LIN {X 0,Y 396.869,Z 754.99,A -85,B 0,C 180,E1 -11238.248,E2 -11238.248} C_VEL
LIN {X 0,Y 396.346,Z 761.62,A -85,B 0,C 180,E1 -11239.785,E2 -11239.785} C_VEL
LIN {X 0,Y 396.097,Z 767.09,A -85,B 0,C 180,E1 -11241.324,E2 -11241.324} C_VEL
LIN {X 0,Y 395.954,Z 771.54,A -85,B 0,C 180,E1 -11242.861,E2 -11242.861} C_VEL
LIN {X 0,Y 395.896,Z 776.01,A -85,B 0,C 180,E1 -11244.906,E2 -11244.906} C_VEL
LIN {X 0,Y 395.865,Z 778.941,A -85,B 0,C 180,E1 -11246.946,E2 -11246.946} C_VEL
LIN {X 0,Y 395.918,Z 779.858,A -85,B 0,C 180,E1 -11247.964,E2 -11247.964} C_VEL
LIN {X 0,Y 395.862,Z 780.59,A -85,B 0,C 180,E1 -11249.999,E2 -11249.999} C_VEL
LIN {X 0,Y 395.918,Z 779.857,A -85,B 0,C 180,E1 -11252.033,E2 -11252.033} C_VEL
LIN {X 0,Y 395.821,Z 777.659,A -85,B 0,C 180,E1 -11254.071,E2 -11254.071} C_VEL
LIN {X 0,Y 395.873,Z 775.066,A -85,B 0,C 180,E1 -11255.602,E2 -11255.602} C_VEL
LIN {X 0,Y 395.952,Z 771.533,A -85,B 0,C 180,E1 -11257.136,E2 -11257.136} C_VEL
LIN {X 0,Y 396.164,Z 765.395,A -85,B 0,C 180,E1 -11259.186,E2 -11259.186} C_VEL
LIN {X 0,Y 396.601,Z 758.452,A -85,B 0,C 180,E1 -11260.98,E2 -11260.98} C_VEL
LIN {X 0,Y 397.107,Z 751.156,A -85,B 0,C 180,E1 -11262.52,E2 -11262.52} C_VEL
LIN {X 0,Y 397.762,Z 742.533,A -85,B 0,C 180,E1 -11264.033,E2 -11264.033} C_VEL
LIN {X 0,Y 398.669,Z 731.702,A -85,B 0,C 180,E1 -11265.594,E2 -11265.594} C_VEL
LIN {X 0,Y 399.641,Z 720.961,A -85,B 0,C 180,E1 -11266.866,E2 -11266.866} C_VEL
LIN {X 0,Y 400.621,Z 709.248,A -85,B 0,C 180,E1 -11268.009,E2 -11268.009} C_VEL
LIN {X 0,Y 401.651,Z 696.152,A -85,B 0,C 180,E1 -11269.036,E2 -11269.036} C_VEL
LIN {X 0,Y 402.545,Z 683.072,A -85,B 0,C 180,E1 -11269.836,E2 -11269.836} C_VEL
LIN {X 0,Y 403.393,Z 668.569,A -85,B 0,C 180,E1 -11270.49,E2 -11270.49} C_VEL
LIN {X 0,Y 404.043,Z 653.982,A -85,B 0,C 180,E1 -11270.922,E2 -11270.922} C_VEL
LIN {X 0,Y 405.933,Z 549.182,A -85,B 0,C 180,E1 -11272.925,E2 -11272.925} C_VEL
LIN {X 0,Y 402.002,Z 522.148,A -85,B 0,C 180,E1 -11273.708,E2 -11273.708} C_VEL
LIN {X 0,Y 403.986,Z 502.582,A -85,B 0,C 180,E1 -11276.89,E2 -11276.89} C_VEL
LIN {X 0,Y 403.831,Z 499.437,A -85,B 0,C 180,E1 -11277.431,E2 -11277.431} C_VEL
LIN {X 0,Y 400.668,Z 486.023,A -85,B 0,C 180,E1 -11279.97,E2 -11279.97} C_VEL
LIN {X 0,Y 397.108,Z 472.647,A -85,B 0,C 180,E1 -11282.667,E2 -11282.667} C_VEL
LIN {X 0,Y 397.103,Z 472.629,A -85,B 0,C 180,E1 -11285.733,E2 -11285.733} C_VEL
LIN {X 0,Y 397.11,Z 472.644,A -85,B 0,C 180,E1 -11289.575,E2 -11289.575} C_VEL
LIN {X 0,Y 397.151,Z 472.639,A -85,B 0,C 180,E1 -11292.254,E2 -11292.254} C_VEL
LIN {X 0,Y 397.143,Z 472.639,A -85,B 0,C 180,E1 -11295.058,E2 -11295.058} C_VEL
LIN {X 0,Y 397.148,Z 472.634,A -85,B 0,C 180,E1 -11298.005,E2 -11298.005} C_VEL
LIN {X 0,Y 397.101,Z 472.639,A -85,B 0,C 180,E1 -11301.725,E2 -11301.725} C_VEL
LIN {X 0,Y 397.116,Z 472.634,A -85,B 0,C 180,E1 -11305.506,E2 -11305.506} C_VEL
LIN {X 0,Y 397.078,Z 472.645,A -85,B 0,C 180,E1 -11309.118,E2 -11309.118} C_VEL
LIN {X 0,Y 397.184,Z 472.632,A -85,B 0,C 180,E1 -11312.609,E2 -11312.609} C_VEL
LIN {X 0,Y 397.122,Z 472.637,A -85,B 0,C 180,E1 -11315.981,E2 -11315.981} C_VEL
LIN {X 0,Y 397.127,Z 472.63,A -85,B 0,C 180,E1 -11319.704,E2 -11319.704} C_VEL
LIN {X 0,Y 397.17,Z 472.635,A -85,B 0,C 180,E1 -11322.844,E2 -11322.844} C_VEL
LIN {X 0,Y 397.215,Z 472.633,A -85,B 0,C 180,E1 -11326.679,E2 -11326.679} C_VEL
LIN {X 0,Y 397.219,Z 472.625,A -85,B 0,C 180,E1 -11329.809,E2 -11329.809} C_VEL
LIN {X 0,Y 397.353,Z 472.606,A -85,B 0,C 180,E1 -11332.888,E2 -11332.888} C_VEL
LIN {X 0,Y 397.247,Z 472.628,A -85,B 0,C 180,E1 -11334.925,E2 -11334.925} C_VEL
LIN {X 0,Y 397.441,Z 472.598,A -85,B 0,C 180,E1 -11337.973,E2 -11337.973} C_VEL
LIN {X 0,Y 397.571,Z 472.582,A -85,B 0,C 180,E1 -11340,E2 -11340} C_VEL
LIN {X 0,Y 397.372,Z 472.602,A -85,B 0,C 180,E1 -11343.042,E2 -11343.042} C_VEL
LIN {X 0,Y 397.352,Z 472.609,A -85,B 0,C 180,E1 -11347.112,E2 -11347.112} C_VEL
LIN {X 0,Y 397.218,Z 472.628,A -85,B 0,C 180,E1 -11350.191,E2 -11350.191} C_VEL
LIN {X 0,Y 397.215,Z 472.622,A -85,B 0,C 180,E1 -11353.322,E2 -11353.322} C_VEL
LIN {X 0,Y 397.16,Z 472.639,A -85,B 0,C 180,E1 -11356.447,E2 -11356.447} C_VEL
LIN {X 0,Y 397.138,Z 472.638,A -85,B 0,C 180,E1 -11359.648,E2 -11359.648} C_VEL
LIN {X 0,Y 397.125,Z 472.64,A -85,B 0,C 180,E1 -11363.041,E2 -11363.041} C_VEL
LIN {X 0,Y 397.125,Z 472.639,A -85,B 0,C 180,E1 -11366.259,E2 -11366.259} C_VEL
LIN {X 0,Y 397.118,Z 472.645,A -85,B 0,C 180,E1 -11368.544,E2 -11368.544} C_VEL
LIN {X 0,Y 397.103,Z 472.644,A -85,B 0,C 180,E1 -11372.07,E2 -11372.07} C_VEL
LIN {X 0,Y 397.112,Z 472.642,A -85,B 0,C 180,E1 -11375.505,E2 -11375.505} C_VEL
LIN {X 0,Y 397.13,Z 472.643,A -85,B 0,C 180,E1 -11378.864,E2 -11378.864} C_VEL
LIN {X 0,Y 397.107,Z 472.648,A -85,B 0,C 180,E1 -11382.263,E2 -11382.263} C_VEL
LIN {X 0,Y 397.159,Z 472.639,A -85,B 0,C 180,E1 -11386.362,E2 -11386.362} C_VEL
LIN {X 0,Y 397.119,Z 472.642,A -85,B 0,C 180,E1 -11389.552,E2 -11389.552} C_VEL
LIN {X 0,Y 397.095,Z 472.637,A -85,B 0,C 180,E1 -11392.791,E2 -11392.791} C_VEL
LIN {X 0,Y 397.115,Z 472.638,A -85,B 0,C 180,E1 -11396.283,E2 -11396.283} C_VEL
LIN {X 0,Y 397.141,Z 472.768,A -85,B 0,C 180,E1 -11399.814,E2 -11399.814} C_VEL
LIN {X 0,Y 400.185,Z 485.268,A -85,B 0,C 180,E1 -11402.833,E2 -11402.833} C_VEL
LIN {X 0,Y 402.101,Z 495.614,A -85,B 0,C 180,E1 -11405.2,E2 -11405.2} C_VEL
LIN {X 0,Y 401.021,Z 508.757,A -85,B 0,C 180,E1 -11407.867,E2 -11407.867} C_VEL
LIN {X 0,Y 400.417,Z 516.355,A -85,B 0,C 180,E1 -11409.385,E2 -11409.385} C_VEL
LIN {X 0,Y 405.174,Z 540.917,A -85,B 0,C 180,E1 -11410.097,E2 -11410.097} C_VEL
LIN {X 0,Y 404.272,Z 629.333,A -85,B 0,C 180,E1 -11411.57,E2 -11411.57} C_VEL
LIN {X 0,Y 403.876,Z 642.226,A -85,B 0,C 180,E1 -11411.977,E2 -11411.977} C_VEL
LIN {X 0,Y 403.222,Z 654.725,A -85,B 0,C 180,E1 -11412.57,E2 -11412.57} C_VEL
LIN {X 0,Y 402.549,Z 665.462,A -85,B 0,C 180,E1 -11413.259,E2 -11413.259} C_VEL
LIN {X 0,Y 401.772,Z 675.831,A -85,B 0,C 180,E1 -11414.106,E2 -11414.106} C_VEL
LIN {X 0,Y 400.872,Z 686.063,A -85,B 0,C 180,E1 -11415.145,E2 -11415.145} C_VEL
LIN {X 0,Y 399.93,Z 695.158,A -85,B 0,C 180,E1 -11416.278,E2 -11416.278} C_VEL
LIN {X 0,Y 399.111,Z 703.472,A -85,B 0,C 180,E1 -11417.544,E2 -11417.544} C_VEL
LIN {X 0,Y 398.218,Z 711.583,A -85,B 0,C 180,E1 -11419.065,E2 -11419.065} C_VEL
LIN {X 0,Y 397.331,Z 719.107,A -85,B 0,C 180,E1 -11420.841,E2 -11420.841} C_VEL
LIN {X 0,Y 396.808,Z 724.17,A -85,B 0,C 180,E1 -11422.368,E2 -11422.368} C_VEL
LIN {X 0,Y 396.438,Z 728.134,A -85,B 0,C 180,E1 -11423.895,E2 -11423.895} C_VEL
LIN {X 0,Y 396.211,Z 730.253,A -85,B 0,C 180,E1 -11424.913,E2 -11424.913} C_VEL
LIN {X 0,Y 396.23,Z 731.923,A -85,B 0,C 180,E1 -11425.933,E2 -11425.933} C_VEL
LIN {X 0,Y 395.984,Z 734.125,A -85,B 0,C 180,E1 -11427.967,E2 -11427.967} C_VEL
LIN {X 0,Y 395.877,Z 734.902,A -85,B 0,C 180,E1 -11430.001,E2 -11430.001} C_VEL
LIN {X 0,Y 395.988,Z 734.15,A -85,B 0,C 180,E1 -11432.085,E2 -11432.085} C_VEL
LIN {X 0,Y 395.386,Z 733.489,A -85,B 0,C 180,E1 -11432.928,E2 -11432.928} C_VEL
LIN {X 0,Y 392.639,Z 732.001,A -85,B 0,C 180,E1 -11434.296,E2 -11434.296} C_VEL
LIN {X 0,Y 390.363,Z 730.358,A -85,B 0,C 180,E1 -11435.388,E2 -11435.388} C_VEL
LIN {X 0,Y 389.488,Z 728.759,A -85,B 0,C 180,E1 -11436.217,E2 -11436.217} C_VEL
LIN {X 0,Y 389.473,Z 728.134,A -85,B 0,C 180,E1 -11436.494,E2 -11436.494} C_VEL
LIN {X 0,Y 389.917,Z 723.331,A -85,B 0,C 180,E1 -11438.292,E2 -11438.292} C_VEL
LIN {X 0,Y 390.69,Z 716.937,A -85,B 0,C 180,E1 -11440.103,E2 -11440.103} C_VEL
LIN {X 0,Y 391.491,Z 709.979,A -85,B 0,C 180,E1 -11441.653,E2 -11441.653} C_VEL
LIN {X 0,Y 392.369,Z 701.359,A -85,B 0,C 180,E1 -11443.203,E2 -11443.203} C_VEL
LIN {X 0,Y 393.541,Z 691.551,A -85,B 0,C 180,E1 -11444.612,E2 -11444.612} C_VEL
LIN {X 0,Y 394.567,Z 680.463,A -85,B 0,C 180,E1 -11445.877,E2 -11445.877} C_VEL
LIN {X 0,Y 395.596,Z 668.922,A -85,B 0,C 180,E1 -11446.914,E2 -11446.914} C_VEL
LIN {X 0,Y 396.493,Z 657.025,A -85,B 0,C 180,E1 -11447.739,E2 -11447.739} C_VEL
LIN {X 0,Y 397.148,Z 644.521,A -85,B 0,C 180,E1 -11448.375,E2 -11448.375} C_VEL
LIN {X 0,Y 397.611,Z 631.502,A -85,B 0,C 180,E1 -11448.82,E2 -11448.82} C_VEL
LIN {X 0,Y 397.959,Z 606.83,A -85,B 0,C 180,E1 -11449.271,E2 -11449.271} C_VEL
LIN {X 0,Y 398.517,Z 540.974,A -85,B 0,C 180,E1 -11450.379,E2 -11450.379} C_VEL
LIN {X 0,Y 393.657,Z 516.432,A -85,B 0,C 180,E1 -11451.114,E2 -11451.114} C_VEL
LIN {X 0,Y 394.865,Z 501.461,A -85,B 0,C 180,E1 -11454.166,E2 -11454.166} C_VEL
LIN {X 0,Y 395.161,Z 496.26,A -85,B 0,C 180,E1 -11455.269,E2 -11455.269} C_VEL
LIN {X 0,Y 392.732,Z 484.528,A -85,B 0,C 180,E1 -11458.035,E2 -11458.035} C_VEL
LIN {X 0,Y 390.068,Z 473.528,A -85,B 0,C 180,E1 -11460.785,E2 -11460.785} C_VEL
LIN {X 0,Y 390.074,Z 473.52,A -85,B 0,C 180,E1 -11464.025,E2 -11464.025} C_VEL
LIN {X 0,Y 390.052,Z 473.527,A -85,B 0,C 180,E1 -11467.552,E2 -11467.552} C_VEL
LIN {X 0,Y 390.064,Z 473.52,A -85,B 0,C 180,E1 -11470.822,E2 -11470.822} C_VEL
LIN {X 0,Y 390.063,Z 473.518,A -85,B 0,C 180,E1 -11473.887,E2 -11473.887} C_VEL
LIN {X 0,Y 390.063,Z 473.52,A -85,B 0,C 180,E1 -11476.79,E2 -11476.79} C_VEL
LIN {X 0,Y 390.062,Z 473.523,A -85,B 0,C 180,E1 -11479.561,E2 -11479.561} C_VEL
LIN {X 0,Y 390.05,Z 473.516,A -85,B 0,C 180,E1 -11482.449,E2 -11482.449} C_VEL
LIN {X 0,Y 390.091,Z 473.52,A -85,B 0,C 180,E1 -11486.047,E2 -11486.047} C_VEL
LIN {X 0,Y 390.053,Z 473.526,A -85,B 0,C 180,E1 -11489.869,E2 -11489.869} C_VEL
LIN {X 0,Y 390.126,Z 473.597,A -85,B 0,C 180,E1 -11490.415,E2 -11490.415} C_VEL
LIN {X 0,Y 393.506,Z 488.852,A -85,B 0,C 180,E1 -11493.254,E2 -11493.254} C_VEL
LIN {X 0,Y 394.678,Z 495.242,A -85,B 0,C 180,E1 -11494.417,E2 -11494.417} C_VEL
LIN {X 0,Y 393.714,Z 514.791,A -85,B 0,C 180,E1 -11497.708,E2 -11497.708} C_VEL
LIN {X 0,Y 393.02,Z 529.732,A -85,B 0,C 180,E1 -11500.217,E2 -11500.217} C_VEL
LIN {X 0,Y 396.012,Z 549.691,A -85,B 0,C 180,E1 -11500.823,E2 -11500.823} C_VEL
LIN {X 0,Y 394.038,Z 641.02,A -85,B 0,C 180,E1 -11502.885,E2 -11502.885} C_VEL
LIN {X 0,Y 393.714,Z 653.198,A -85,B 0,C 180,E1 -11503.338,E2 -11503.338} C_VEL
LIN {X 0,Y 393.126,Z 666.44,A -85,B 0,C 180,E1 -11504.046,E2 -11504.046} C_VEL
LIN {X 0,Y 392.539,Z 677.977,A -85,B 0,C 180,E1 -11504.86,E2 -11504.86} C_VEL
LIN {X 0,Y 391.975,Z 688.733,A -85,B 0,C 180,E1 -11505.823,E2 -11505.823} C_VEL
LIN {X 0,Y 391.293,Z 699.539,A -85,B 0,C 180,E1 -11507.026,E2 -11507.026} C_VEL
LIN {X 0,Y 390.633,Z 709.04,A -85,B 0,C 180,E1 -11508.322,E2 -11508.322} C_VEL
LIN {X 0,Y 390.037,Z 718.2,A -85,B 0,C 180,E1 -11509.881,E2 -11509.881} C_VEL
LIN {X 0,Y 389.558,Z 725.574,A -85,B 0,C 180,E1 -11511.44,E2 -11511.44} C_VEL
LIN {X 0,Y 389.267,Z 730.534,A -85,B 0,C 180,E1 -11512.739,E2 -11512.739} C_VEL
LIN {X 0,Y 389.075,Z 735.328,A -85,B 0,C 180,E1 -11514.298,E2 -11514.298} C_VEL
LIN {X 0,Y 388.873,Z 738.948,A -85,B 0,C 180,E1 -11515.854,E2 -11515.854} C_VEL
LIN {X 0,Y 388.855,Z 740.743,A -85,B 0,C 180,E1 -11516.892,E2 -11516.892} C_VEL
LIN {X 0,Y 388.834,Z 742.115,A -85,B 0,C 180,E1 -11517.928,E2 -11517.928} C_VEL
LIN {X 0,Y 388.767,Z 743.07,A -85,B 0,C 180,E1 -11518.964,E2 -11518.964} C_VEL
LIN {X 0,Y 388.748,Z 743.551,A -85,B 0,C 180,E1 -11520,E2 -11520} C_VEL
LIN {X 0,Y 388.787,Z 743.621,A -85,B 0,C 180,E1 -11521.036,E2 -11521.036} C_VEL
LIN {X 0,Y 388.874,Z 743.279,A -85,B 0,C 180,E1 -11522.071,E2 -11522.071} C_VEL
LIN {X 0,Y 389.015,Z 742.463,A -85,B 0,C 180,E1 -11523.107,E2 -11523.107} C_VEL
LIN {X 0,Y 389.091,Z 741.23,A -85,B 0,C 180,E1 -11524.143,E2 -11524.143} C_VEL
LIN {X 0,Y 389.194,Z 738.55,A -85,B 0,C 180,E1 -11525.7,E2 -11525.7} C_VEL
LIN {X 0,Y 389.568,Z 734.781,A -85,B 0,C 180,E1 -11527.255,E2 -11527.255} C_VEL
LIN {X 0,Y 389.993,Z 729.855,A -85,B 0,C 180,E1 -11528.811,E2 -11528.811} C_VEL
LIN {X 0,Y 390.649,Z 723.594,A -85,B 0,C 180,E1 -11530.364,E2 -11530.364} C_VEL
LIN {X 0,Y 391.342,Z 715.749,A -85,B 0,C 180,E1 -11531.919,E2 -11531.919} C_VEL
LIN {X 0,Y 392.056,Z 707.734,A -85,B 0,C 180,E1 -11533.212,E2 -11533.212} C_VEL
LIN {X 0,Y 392.976,Z 697.935,A -85,B 0,C 180,E1 -11534.5,E2 -11534.5} C_VEL
LIN {X 0,Y 394.037,Z 685.631,A -85,B 0,C 180,E1 -11535.783,E2 -11535.783} C_VEL
LIN {X 0,Y 394.787,Z 674.799,A -85,B 0,C 180,E1 -11536.682,E2 -11536.682} C_VEL
LIN {X 0,Y 395.579,Z 662.942,A -85,B 0,C 180,E1 -11537.446,E2 -11537.446} C_VEL
LIN {X 0,Y 396.221,Z 649.645,A -85,B 0,C 180,E1 -11538.084,E2 -11538.084} C_VEL
LIN {X 0,Y 396.743,Z 635.325,A -85,B 0,C 180,E1 -11538.527,E2 -11538.527} C_VEL
LIN {X 0,Y 399.017,Z 569.961,A -85,B 0,C 180,E1 -11540.177,E2 -11540.177} C_VEL
LIN {X 0,Y 399.7,Z 550.541,A -85,B 0,C 180,E1 -11540.697,E2 -11540.697} C_VEL
LIN {X 0,Y 397.165,Z 537.555,A -85,B 0,C 180,E1 -11541.299,E2 -11541.299} C_VEL
LIN {X 0,Y 396.171,Z 533.316,A -85,B 0,C 180,E1 -11541.53,E2 -11541.53} C_VEL
LIN {X 0,Y 397.739,Z 510.589,A -85,B 0,C 180,E1 -11545.379,E2 -11545.379} C_VEL
LIN {X 0,Y 398.225,Z 502.569,A -85,B 0,C 180,E1 -11546.746,E2 -11546.746} C_VEL
LIN {X 0,Y 397.063,Z 495.233,A -85,B 0,C 180,E1 -11548.217,E2 -11548.217} C_VEL
LIN {X 0,Y 394.529,Z 486.198,A -85,B 0,C 180,E1 -11550.183,E2 -11550.183} C_VEL
LIN {X 0,Y 391.296,Z 476.89,A -85,B 0,C 180,E1 -11552.416,E2 -11552.416} C_VEL
LIN {X 0,Y 390.097,Z 473.519,A -85,B 0,C 180,E1 -11553.332,E2 -11553.332} C_VEL
LIN {X 0,Y 390.065,Z 473.525,A -85,B 0,C 180,E1 -11556.483,E2 -11556.483} C_VEL
LIN {X 0,Y 390.077,Z 473.52,A -85,B 0,C 180,E1 -11559.218,E2 -11559.218} C_VEL
LIN {X 0,Y 390.047,Z 473.525,A -85,B 0,C 180,E1 -11562.373,E2 -11562.373} C_VEL
LIN {X 0,Y 390.049,Z 473.523,A -85,B 0,C 180,E1 -11565.354,E2 -11565.354} C_VEL
LIN {X 0,Y 390.036,Z 473.526,A -85,B 0,C 180,E1 -11568.186,E2 -11568.186} C_VEL
LIN {X 0,Y 390.092,Z 473.515,A -85,B 0,C 180,E1 -11570.907,E2 -11570.907} C_VEL
LIN {X 0,Y 390.089,Z 473.52,A -85,B 0,C 180,E1 -11574.792,E2 -11574.792} C_VEL
LIN {X 0,Y 390.078,Z 473.534,A -85,B 0,C 180,E1 -11576.858,E2 -11576.858} C_VEL
LIN {X 0,Y 394.193,Z 489.099,A -85,B 0,C 180,E1 -11580.051,E2 -11580.051} C_VEL
LIN {X 0,Y 396.925,Z 500.672,A -85,B 0,C 180,E1 -11582.289,E2 -11582.289} C_VEL
LIN {X 0,Y 397.307,Z 502.415,A -85,B 0,C 180,E1 -11582.617,E2 -11582.617} C_VEL
LIN {X 0,Y 395.596,Z 519.085,A -85,B 0,C 180,E1 -11585.378,E2 -11585.378} C_VEL
LIN {X 0,Y 395.25,Z 522.317,A -85,B 0,C 180,E1 -11585.915,E2 -11585.915} C_VEL
LIN {X 0,Y 399.311,Z 550.056,A -85,B 0,C 180,E1 -11586.712,E2 -11586.712} C_VEL
LIN {X 0,Y 397.368,Z 652.886,A -85,B 0,C 180,E1 -11588.707,E2 -11588.707} C_VEL
LIN {X 0,Y 396.788,Z 666.902,A -85,B 0,C 180,E1 -11589.116,E2 -11589.116} C_VEL
LIN {X 0,Y 395.894,Z 681.293,A -85,B 0,C 180,E1 -11589.746,E2 -11589.746} C_VEL
LIN {X 0,Y 394.988,Z 694.805,A -85,B 0,C 180,E1 -11590.566,E2 -11590.566} C_VEL
LIN {X 0,Y 394.005,Z 707.301,A -85,B 0,C 180,E1 -11591.541,E2 -11591.541} C_VEL
LIN {X 0,Y 392.907,Z 719.288,A -85,B 0,C 180,E1 -11592.699,E2 -11592.699} C_VEL
LIN {X 0,Y 391.778,Z 731.243,A -85,B 0,C 180,E1 -11594.122,E2 -11594.122} C_VEL
LIN {X 0,Y 390.79,Z 742.088,A -85,B 0,C 180,E1 -11595.709,E2 -11595.709} C_VEL
LIN {X 0,Y 390.155,Z 750.762,A -85,B 0,C 180,E1 -11597.258,E2 -11597.258} C_VEL
LIN {X 0,Y 389.473,Z 759.092,A -85,B 0,C 180,E1 -11599.077,E2 -11599.077} C_VEL
LIN {X 0,Y 389.098,Z 764.977,A -85,B 0,C 180,E1 -11600.643,E2 -11600.643} C_VEL
LIN {X 0,Y 388.896,Z 769.755,A -85,B 0,C 180,E1 -11602.209,E2 -11602.209} C_VEL
LIN {X 0,Y 388.789,Z 774.38,A -85,B 0,C 180,E1 -11604.157,E2 -11604.157} C_VEL
LIN {X 0,Y 388.745,Z 777.246,A -85,B 0,C 180,E1 -11605.852,E2 -11605.852} C_VEL
LIN {X 0,Y 388.849,Z 779.449,A -85,B 0,C 180,E1 -11607.927,E2 -11607.927} C_VEL
LIN {X 0,Y 388.787,Z 780.181,A -85,B 0,C 180,E1 -11609.999,E2 -11609.999} C_VEL
LIN {X 0,Y 388.848,Z 779.448,A -85,B 0,C 180,E1 -11612.07,E2 -11612.07} C_VEL
LIN {X 0,Y 388.744,Z 777.246,A -85,B 0,C 180,E1 -11614.146,E2 -11614.146} C_VEL
LIN {X 0,Y 388.788,Z 774.375,A -85,B 0,C 180,E1 -11615.841,E2 -11615.841} C_VEL
LIN {X 0,Y 388.893,Z 769.744,A -85,B 0,C 180,E1 -11617.788,E2 -11617.788} C_VEL
LIN {X 0,Y 389.095,Z 764.964,A -85,B 0,C 180,E1 -11619.354,E2 -11619.354} C_VEL
LIN {X 0,Y 389.573,Z 758.009,A -85,B 0,C 180,E1 -11621.181,E2 -11621.181} C_VEL
LIN {X 0,Y 390.177,Z 749.536,A -85,B 0,C 180,E1 -11622.968,E2 -11622.968} C_VEL
LIN {X 0,Y 390.963,Z 740.229,A -85,B 0,C 180,E1 -11624.575,E2 -11624.575} C_VEL
LIN {X 0,Y 391.792,Z 731.211,A -85,B 0,C 180,E1 -11625.874,E2 -11625.874} C_VEL
LIN {X 0,Y 392.807,Z 720.442,A -85,B 0,C 180,E1 -11627.169,E2 -11627.169} C_VEL
LIN {X 0,Y 393.838,Z 708.693,A -85,B 0,C 180,E1 -11628.33,E2 -11628.33} C_VEL
LIN {X 0,Y 394.87,Z 695.851,A -85,B 0,C 180,E1 -11629.352,E2 -11629.352} C_VEL
LIN {X 0,Y 395.862,Z 682.385,A -85,B 0,C 180,E1 -11630.185,E2 -11630.185} C_VEL
LIN {X 0,Y 396.733,Z 667.646,A -85,B 0,C 180,E1 -11630.85,E2 -11630.85} C_VEL
LIN {X 0,Y 397.344,Z 654.089,A -85,B 0,C 180,E1 -11631.258,E2 -11631.258} C_VEL
LIN {X 0,Y 399.311,Z 549.835,A -85,B 0,C 180,E1 -11633.282,E2 -11633.282} C_VEL
LIN {X 0,Y 395.271,Z 522.131,A -85,B 0,C 180,E1 -11634.099,E2 -11634.099} C_VEL
LIN {X 0,Y 397.21,Z 504.027,A -85,B 0,C 180,E1 -11637.102,E2 -11637.102} C_VEL
LIN {X 0,Y 396.904,Z 500.649,A -85,B 0,C 180,E1 -11637.705,E2 -11637.705} C_VEL
LIN {X 0,Y 393.389,Z 485.818,A -85,B 0,C 180,E1 -11640.585,E2 -11640.585} C_VEL
LIN {X 0,Y 390.072,Z 473.522,A -85,B 0,C 180,E1 -11643.178,E2 -11643.178} C_VEL
LIN {X 0,Y 390.054,Z 473.517,A -85,B 0,C 180,E1 -11646.482,E2 -11646.482} C_VEL
LIN {X 0,Y 390.068,Z 473.52,A -85,B 0,C 180,E1 -11649.218,E2 -11649.218} C_VEL
LIN {X 0,Y 390.113,Z 473.516,A -85,B 0,C 180,E1 -11652.385,E2 -11652.385} C_VEL
LIN {X 0,Y 390.121,Z 473.511,A -85,B 0,C 180,E1 -11656.101,E2 -11656.101} C_VEL
LIN {X 0,Y 390.07,Z 473.515,A -85,B 0,C 180,E1 -11659.562,E2 -11659.562} C_VEL
LIN {X 0,Y 390.038,Z 473.518,A -85,B 0,C 180,E1 -11662.447,E2 -11662.447} C_VEL
LIN {X 0,Y 390.058,Z 473.514,A -85,B 0,C 180,E1 -11666.044,E2 -11666.044} C_VEL
LIN {X 0,Y 390.038,Z 473.521,A -85,B 0,C 180,E1 -11668.497,E2 -11668.497} C_VEL
LIN {X 0,Y 390.107,Z 473.512,A -85,B 0,C 180,E1 -11672.069,E2 -11672.069} C_VEL
LIN {X 0,Y 390.069,Z 473.515,A -85,B 0,C 180,E1 -11675.519,E2 -11675.519} C_VEL
LIN {X 0,Y 390.044,Z 473.503,A -85,B 0,C 180,E1 -11678.877,E2 -11678.877} C_VEL
LIN {X 0,Y 390.117,Z 473.515,A -85,B 0,C 180,E1 -11682.166,E2 -11682.166} C_VEL
LIN {X 0,Y 390.136,Z 473.51,A -85,B 0,C 180,E1 -11685.392,E2 -11685.392} C_VEL
LIN {X 0,Y 390.15,Z 473.506,A -85,B 0,C 180,E1 -11688.571,E2 -11688.571} C_VEL
LIN {X 0,Y 390.332,Z 473.487,A -85,B 0,C 180,E1 -11691.993,E2 -11691.993} C_VEL
LIN {X 0,Y 390.219,Z 473.502,A -85,B 0,C 180,E1 -11694.834,E2 -11694.834} C_VEL
LIN {X 0,Y 390.41,Z 473.473,A -85,B 0,C 180,E1 -11697.937,E2 -11697.937} C_VEL
LIN {X 0,Y 390.541,Z 473.458,A -85,B 0,C 180,E1 -11700,E2 -11700} C_VEL
LIN {X 0,Y 390.306,Z 473.482,A -85,B 0,C 180,E1 -11703.097,E2 -11703.097} C_VEL
LIN {X 0,Y 390.298,Z 473.489,A -85,B 0,C 180,E1 -11706.653,E2 -11706.653} C_VEL
LIN {X 0,Y 390.199,Z 473.5,A -85,B 0,C 180,E1 -11709.329,E2 -11709.329} C_VEL
LIN {X 0,Y 390.167,Z 473.505,A -85,B 0,C 180,E1 -11712.483,E2 -11712.483} C_VEL
LIN {X 0,Y 390.134,Z 473.511,A -85,B 0,C 180,E1 -11715.677,E2 -11715.677} C_VEL
LIN {X 0,Y 390.095,Z 473.518,A -85,B 0,C 180,E1 -11718.923,E2 -11718.923} C_VEL
LIN {X 0,Y 390.03,Z 473.521,A -85,B 0,C 180,E1 -11722.235,E2 -11722.235} C_VEL
LIN {X 0,Y 390.109,Z 473.512,A -85,B 0,C 180,E1 -11725.744,E2 -11725.744} C_VEL
LIN {X 0,Y 390.056,Z 473.519,A -85,B 0,C 180,E1 -11729.11,E2 -11729.11} C_VEL
LIN {X 0,Y 390.047,Z 473.522,A -85,B 0,C 180,E1 -11732.721,E2 -11732.721} C_VEL
LIN {X 0,Y 390.049,Z 473.523,A -85,B 0,C 180,E1 -11735.827,E2 -11735.827} C_VEL
LIN {X 0,Y 390.067,Z 473.52,A -85,B 0,C 180,E1 -11739.221,E2 -11739.221} C_VEL
LIN {X 0,Y 390.073,Z 473.523,A -85,B 0,C 180,E1 -11742.382,E2 -11742.382} C_VEL
LIN {X 0,Y 390.099,Z 473.516,A -85,B 0,C 180,E1 -11746.107,E2 -11746.107} C_VEL
LIN {X 0,Y 390.078,Z 473.52,A -85,B 0,C 180,E1 -11749.175,E2 -11749.175} C_VEL
LIN {X 0,Y 390.043,Z 473.518,A -85,B 0,C 180,E1 -11752.45,E2 -11752.45} C_VEL
LIN {X 0,Y 390.08,Z 473.514,A -85,B 0,C 180,E1 -11756.048,E2 -11756.048} C_VEL
LIN {X 0,Y 390.072,Z 473.593,A -85,B 0,C 180,E1 -11759.368,E2 -11759.368} C_VEL
LIN {X 0,Y 393.284,Z 486.581,A -85,B 0,C 180,E1 -11762.571,E2 -11762.571} C_VEL
LIN {X 0,Y 395.258,Z 497.309,A -85,B 0,C 180,E1 -11765.07,E2 -11765.07} C_VEL
LIN {X 0,Y 394.135,Z 510.26,A -85,B 0,C 180,E1 -11767.735,E2 -11767.735} C_VEL
LIN {X 0,Y 393.621,Z 516.406,A -85,B 0,C 180,E1 -11768.982,E2 -11768.982} C_VEL
LIN {X 0,Y 398.641,Z 542.404,A -85,B 0,C 180,E1 -11769.752,E2 -11769.752} C_VEL
LIN {X 0,Y 397.624,Z 629.27,A -85,B 0,C 180,E1 -11771.217,E2 -11771.217} C_VEL
LIN {X 0,Y 397.211,Z 642.287,A -85,B 0,C 180,E1 -11771.631,E2 -11771.631} C_VEL
LIN {X 0,Y 396.491,Z 655.415,A -85,B 0,C 180,E1 -11772.264,E2 -11772.264} C_VEL
LIN {X 0,Y 395.722,Z 667.788,A -85,B 0,C 180,E1 -11773.095,E2 -11773.095} C_VEL
LIN {X 0,Y 394.827,Z 678.149,A -85,B 0,C 180,E1 -11773.991,E2 -11773.991} C_VEL
LIN {X 0,Y 393.806,Z 688.712,A -85,B 0,C 180,E1 -11775.137,E2 -11775.137} C_VEL
LIN {X 0,Y 392.625,Z 699.133,A -85,B 0,C 180,E1 -11776.545,E2 -11776.545} C_VEL
LIN {X 0,Y 391.809,Z 706.82,A -85,B 0,C 180,E1 -11777.834,E2 -11777.834} C_VEL
LIN {X 0,Y 390.996,Z 714.39,A -85,B 0,C 180,E1 -11779.385,E2 -11779.385} C_VEL
LIN {X 0,Y 390.12,Z 721.344,A -85,B 0,C 180,E1 -11781.193,E2 -11781.193} C_VEL
LIN {X 0,Y 389.617,Z 726.149,A -85,B 0,C 180,E1 -11782.797,E2 -11782.797} C_VEL
LIN {X 0,Y 389.249,Z 729.655,A -85,B 0,C 180,E1 -11784.302,E2 -11784.302} C_VEL
LIN {X 0,Y 389.145,Z 732.336,A -85,B 0,C 180,E1 -11785.859,E2 -11785.859} C_VEL
LIN {X 0,Y 389.068,Z 733.613,A -85,B 0,C 180,E1 -11786.895,E2 -11786.895} C_VEL
LIN {X 0,Y 388.82,Z 735.099,A -85,B 0,C 180,E1 -11788.966,E2 -11788.966} C_VEL
LIN {X 0,Y 388.82,Z 735.14,A -85,B 0,C 180,E1 -11791.037,E2 -11791.037} C_VEL
LIN {X 0,Y 389.061,Z 733.707,A -85,B 0,C 180,E1 -11793.108,E2 -11793.108} C_VEL
LIN {X 0,Y 389.139,Z 730.838,A -85,B 0,C 180,E1 -11795.182,E2 -11795.182} C_VEL
LIN {X 0,Y 389.473,Z 728.134,A -85,B 0,C 180,E1 -11796.494,E2 -11796.494} C_VEL
LIN {X 0,Y 389.031,Z 726.201,A -85,B 0,C 180,E1 -11797.312,E2 -11797.312} C_VEL
LIN {X 0,Y 386.59,Z 722.711,A -85,B 0,C 180,E1 -11798.634,E2 -11798.634} C_VEL
LIN {X 0,Y 384.23,Z 718.625,A -85,B 0,C 180,E1 -11799.931,E2 -11799.931} C_VEL
LIN {X 0,Y 383.922,Z 715.69,A -85,B 0,C 180,E1 -11800.698,E2 -11800.698} C_VEL
LIN {X 0,Y 384.866,Z 707.784,A -85,B 0,C 180,E1 -11802.391,E2 -11802.391} C_VEL
LIN {X 0,Y 385.694,Z 700.216,A -85,B 0,C 180,E1 -11803.704,E2 -11803.704} C_VEL
LIN {X 0,Y 386.934,Z 689.951,A -85,B 0,C 180,E1 -11805.136,E2 -11805.136} C_VEL
LIN {X 0,Y 387.918,Z 679.348,A -85,B 0,C 180,E1 -11806.33,E2 -11806.33} C_VEL
LIN {X 0,Y 388.974,Z 667.896,A -85,B 0,C 180,E1 -11807.346,E2 -11807.346} C_VEL
LIN {X 0,Y 389.831,Z 656.578,A -85,B 0,C 180,E1 -11808.12,E2 -11808.12} C_VEL
LIN {X 0,Y 390.521,Z 643.778,A -85,B 0,C 180,E1 -11808.766,E2 -11808.766} C_VEL
LIN {X 0,Y 390.991,Z 631.407,A -85,B 0,C 180,E1 -11809.185,E2 -11809.185} C_VEL
LIN {X 0,Y 391.327,Z 604.587,A -85,B 0,C 180,E1 -11809.68,E2 -11809.68} C_VEL
LIN {X 0,Y 391.961,Z 542.061,A -85,B 0,C 180,E1 -11810.746,E2 -11810.746} C_VEL
LIN {X 0,Y 386.872,Z 516.455,A -85,B 0,C 180,E1 -11811.539,E2 -11811.539} C_VEL
LIN {X 0,Y 388.172,Z 501.64,A -85,B 0,C 180,E1 -11814.61,E2 -11814.61} C_VEL
LIN {X 0,Y 388.349,Z 498.091,A -85,B 0,C 180,E1 -11815.379,E2 -11815.379} C_VEL
LIN {X 0,Y 385.846,Z 486.056,A -85,B 0,C 180,E1 -11818.268,E2 -11818.268} C_VEL
LIN {X 0,Y 383.262,Z 475.636,A -85,B 0,C 180,E1 -11820.895,E2 -11820.895} C_VEL
LIN {X 0,Y 383.006,Z 474.406,A -85,B 0,C 180,E1 -11821.225,E2 -11821.225} C_VEL
LIN {X 0,Y 383.024,Z 474.398,A -85,B 0,C 180,E1 -11824.669,E2 -11824.669} C_VEL
LIN {X 0,Y 383.008,Z 474.4,A -85,B 0,C 180,E1 -11827.905,E2 -11827.905} C_VEL
LIN {X 0,Y 382.992,Z 474.4,A -85,B 0,C 180,E1 -11831.348,E2 -11831.348} C_VEL
LIN {X 0,Y 383.004,Z 474.395,A -85,B 0,C 180,E1 -11834.304,E2 -11834.304} C_VEL
LIN {X 0,Y 383.016,Z 474.396,A -85,B 0,C 180,E1 -11837.241,E2 -11837.241} C_VEL
LIN {X 0,Y 383.02,Z 474.397,A -85,B 0,C 180,E1 -11840.414,E2 -11840.414} C_VEL
LIN {X 0,Y 383.033,Z 474.399,A -85,B 0,C 180,E1 -11844.045,E2 -11844.045} C_VEL
LIN {X 0,Y 382.993,Z 474.405,A -85,B 0,C 180,E1 -11847.578,E2 -11847.578} C_VEL
LIN {X 0,Y 383.042,Z 474.439,A -85,B 0,C 180,E1 -11850.127,E2 -11850.127} C_VEL
LIN {X 0,Y 386.482,Z 489.74,A -85,B 0,C 180,E1 -11853.006,E2 -11853.006} C_VEL
LIN {X 0,Y 387.748,Z 496.285,A -85,B 0,C 180,E1 -11854.214,E2 -11854.214} C_VEL
LIN {X 0,Y 386.876,Z 514.365,A -85,B 0,C 180,E1 -11857.292,E2 -11857.292} C_VEL
LIN {X 0,Y 386.116,Z 530.078,A -85,B 0,C 180,E1 -11859.946,E2 -11859.946} C_VEL
LIN {X 0,Y 389.1,Z 551.277,A -85,B 0,C 180,E1 -11860.586,E2 -11860.586} C_VEL
LIN {X 0,Y 387.089,Z 640.853,A -85,B 0,C 180,E1 -11862.67,E2 -11862.67} C_VEL
LIN {X 0,Y 386.737,Z 653.842,A -85,B 0,C 180,E1 -11863.164,E2 -11863.164} C_VEL
LIN {X 0,Y 386.14,Z 666.958,A -85,B 0,C 180,E1 -11863.885,E2 -11863.885} C_VEL
LIN {X 0,Y 385.467,Z 679.541,A -85,B 0,C 180,E1 -11864.806,E2 -11864.806} C_VEL
LIN {X 0,Y 384.796,Z 691.372,A -85,B 0,C 180,E1 -11865.925,E2 -11865.925} C_VEL
LIN {X 0,Y 384.168,Z 701.006,A -85,B 0,C 180,E1 -11867.05,E2 -11867.05} C_VEL
LIN {X 0,Y 383.488,Z 710.257,A -85,B 0,C 180,E1 -11868.37,E2 -11868.37} C_VEL
LIN {X 0,Y 382.916,Z 719.281,A -85,B 0,C 180,E1 -11869.958,E2 -11869.958} C_VEL
LIN {X 0,Y 382.443,Z 726.496,A -85,B 0,C 180,E1 -11871.546,E2 -11871.546} C_VEL
LIN {X 0,Y 382.112,Z 732.811,A -85,B 0,C 180,E1 -11873.319,E2 -11873.319} C_VEL
LIN {X 0,Y 381.944,Z 736.704,A -85,B 0,C 180,E1 -11874.721,E2 -11874.721} C_VEL
LIN {X 0,Y 381.799,Z 739.078,A -85,B 0,C 180,E1 -11875.777,E2 -11875.777} C_VEL
LIN {X 0,Y 381.76,Z 740.938,A -85,B 0,C 180,E1 -11876.834,E2 -11876.834} C_VEL
LIN {X 0,Y 381.753,Z 742.35,A -85,B 0,C 180,E1 -11877.89,E2 -11877.89} C_VEL
LIN {X 0,Y 381.7,Z 743.353,A -85,B 0,C 180,E1 -11878.945,E2 -11878.945} C_VEL
LIN {X 0,Y 381.678,Z 743.888,A -85,B 0,C 180,E1 -11880,E2 -11880} C_VEL
LIN {X 0,Y 381.719,Z 743.99,A -85,B 0,C 180,E1 -11881.055,E2 -11881.055} C_VEL
LIN {X 0,Y 381.813,Z 743.681,A -85,B 0,C 180,E1 -11882.11,E2 -11882.11} C_VEL
LIN {X 0,Y 381.961,Z 742.917,A -85,B 0,C 180,E1 -11883.164,E2 -11883.164} C_VEL
LIN {X 0,Y 382.011,Z 741.714,A -85,B 0,C 180,E1 -11884.22,E2 -11884.22} C_VEL
LIN {X 0,Y 382.161,Z 739.101,A -85,B 0,C 180,E1 -11885.805,E2 -11885.805} C_VEL
LIN {X 0,Y 382.555,Z 735.412,A -85,B 0,C 180,E1 -11887.388,E2 -11887.388} C_VEL
LIN {X 0,Y 383.02,Z 730.554,A -85,B 0,C 180,E1 -11888.973,E2 -11888.973} C_VEL
LIN {X 0,Y 383.712,Z 724.374,A -85,B 0,C 180,E1 -11890.554,E2 -11890.554} C_VEL
LIN {X 0,Y 384.455,Z 716.594,A -85,B 0,C 180,E1 -11892.135,E2 -11892.135} C_VEL
LIN {X 0,Y 385.358,Z 706.949,A -85,B 0,C 180,E1 -11893.715,E2 -11893.715} C_VEL
LIN {X 0,Y 386.482,Z 696.456,A -85,B 0,C 180,E1 -11895.068,E2 -11895.068} C_VEL
LIN {X 0,Y 387.443,Z 685.682,A -85,B 0,C 180,E1 -11896.194,E2 -11896.194} C_VEL
LIN {X 0,Y 388.364,Z 672.938,A -85,B 0,C 180,E1 -11897.237,E2 -11897.237} C_VEL
LIN {X 0,Y 389.181,Z 660.423,A -85,B 0,C 180,E1 -11898.014,E2 -11898.014} C_VEL
LIN {X 0,Y 389.931,Z 645.802,A -85,B 0,C 180,E1 -11898.658,E2 -11898.658} C_VEL
LIN {X 0,Y 391.262,Z 607.662,A -85,B 0,C 180,E1 -11899.682,E2 -11899.682} C_VEL
LIN {X 0,Y 393.514,Z 551.711,A -85,B 0,C 180,E1 -11901.178,E2 -11901.178} C_VEL
LIN {X 0,Y 391.231,Z 539.757,A -85,B 0,C 180,E1 -11901.771,E2 -11901.771} C_VEL
LIN {X 0,Y 389.851,Z 533.727,A -85,B 0,C 180,E1 -11902.112,E2 -11902.112} C_VEL
LIN {X 0,Y 391.439,Z 512.102,A -85,B 0,C 180,E1 -11905.831,E2 -11905.831} C_VEL
LIN {X 0,Y 391.907,Z 504.375,A -85,B 0,C 180,E1 -11907.212,E2 -11907.212} C_VEL
LIN {X 0,Y 390.657,Z 497.292,A -85,B 0,C 180,E1 -11908.68,E2 -11908.68} C_VEL
LIN {X 0,Y 387.868,Z 487.536,A -85,B 0,C 180,E1 -11910.91,E2 -11910.91} C_VEL
LIN {X 0,Y 384.548,Z 478.43,A -85,B 0,C 180,E1 -11913.249,E2 -11913.249} C_VEL
LIN {X 0,Y 383.043,Z 474.397,A -85,B 0,C 180,E1 -11914.403,E2 -11914.403} C_VEL
LIN {X 0,Y 383.007,Z 474.403,A -85,B 0,C 180,E1 -11917.904,E2 -11917.904} C_VEL
LIN {X 0,Y 382.989,Z 474.405,A -85,B 0,C 180,E1 -11921.347,E2 -11921.347} C_VEL
LIN {X 0,Y 383.001,Z 474.404,A -85,B 0,C 180,E1 -11924.303,E2 -11924.303} C_VEL
LIN {X 0,Y 383.015,Z 474.398,A -85,B 0,C 180,E1 -11927.239,E2 -11927.239} C_VEL
LIN {X 0,Y 383.018,Z 474.397,A -85,B 0,C 180,E1 -11930.413,E2 -11930.413} C_VEL
LIN {X 0,Y 383.029,Z 474.397,A -85,B 0,C 180,E1 -11934.044,E2 -11934.044} C_VEL
LIN {X 0,Y 383.052,Z 474.408,A -85,B 0,C 180,E1 -11936.37,E2 -11936.37} C_VEL
LIN {X 0,Y 387.306,Z 490.402,A -85,B 0,C 180,E1 -11939.735,E2 -11939.735} C_VEL
LIN {X 0,Y 390.282,Z 503.153,A -85,B 0,C 180,E1 -11942.249,E2 -11942.249} C_VEL
LIN {X 0,Y 390.464,Z 505.506,A -85,B 0,C 180,E1 -11942.678,E2 -11942.678} C_VEL
LIN {X 0,Y 388.526,Z 522.291,A -85,B 0,C 180,E1 -11945.504,E2 -11945.504} C_VEL
LIN {X 0,Y 392.711,Z 550.453,A -85,B 0,C 180,E1 -11946.336,E2 -11946.336} C_VEL
LIN {X 0,Y 390.671,Z 654.466,A -85,B 0,C 180,E1 -11948.393,E2 -11948.393} C_VEL
LIN {X 0,Y 390.015,Z 668.671,A -85,B 0,C 180,E1 -11948.84,E2 -11948.84} C_VEL
LIN {X 0,Y 389.073,Z 682.935,A -85,B 0,C 180,E1 -11949.513,E2 -11949.513} C_VEL
LIN {X 0,Y 388.024,Z 696.825,A -85,B 0,C 180,E1 -11950.406,E2 -11950.406} C_VEL
LIN {X 0,Y 387.006,Z 709.645,A -85,B 0,C 180,E1 -11951.469,E2 -11951.469} C_VEL
LIN {X 0,Y 385.847,Z 721.167,A -85,B 0,C 180,E1 -11952.646,E2 -11952.646} C_VEL
LIN {X 0,Y 384.692,Z 732.723,A -85,B 0,C 180,E1 -11954.094,E2 -11954.094} C_VEL
LIN {X 0,Y 383.715,Z 743.02,A -85,B 0,C 180,E1 -11955.683,E2 -11955.683} C_VEL
LIN {X 0,Y 383.042,Z 751.56,A -85,B 0,C 180,E1 -11957.279,E2 -11957.279} C_VEL
LIN {X 0,Y 382.354,Z 759.704,A -85,B 0,C 180,E1 -11959.139,E2 -11959.139} C_VEL
LIN {X 0,Y 381.937,Z 766.234,A -85,B 0,C 180,E1 -11961,E2 -11961} C_VEL
LIN {X 0,Y 381.796,Z 770.699,A -85,B 0,C 180,E1 -11962.595,E2 -11962.595} C_VEL
LIN {X 0,Y 381.739,Z 773.456,A -85,B 0,C 180,E1 -11963.807,E2 -11963.807} C_VEL
LIN {X 0,Y 381.67,Z 776.834,A -85,B 0,C 180,E1 -11965.775,E2 -11965.775} C_VEL
LIN {X 0,Y 381.779,Z 779.04,A -85,B 0,C 180,E1 -11967.889,E2 -11967.889} C_VEL
LIN {X 0,Y 381.714,Z 779.773,A -85,B 0,C 180,E1 -11969.999,E2 -11969.999} C_VEL
LIN {X 0,Y 381.779,Z 779.038,A -85,B 0,C 180,E1 -11972.109,E2 -11972.109} C_VEL
LIN {X 0,Y 381.669,Z 776.833,A -85,B 0,C 180,E1 -11974.223,E2 -11974.223} C_VEL
LIN {X 0,Y 381.761,Z 773.134,A -85,B 0,C 180,E1 -11976.34,E2 -11976.34} C_VEL
LIN {X 0,Y 381.89,Z 767.829,A -85,B 0,C 180,E1 -11978.465,E2 -11978.465} C_VEL
LIN {X 0,Y 382.151,Z 762.67,A -85,B 0,C 180,E1 -11980.06,E2 -11980.06} C_VEL
LIN {X 0,Y 382.749,Z 755.255,A -85,B 0,C 180,E1 -11981.92,E2 -11981.92} C_VEL
LIN {X 0,Y 383.403,Z 746.464,A -85,B 0,C 180,E1 -11983.707,E2 -11983.707} C_VEL
LIN {X 0,Y 384.318,Z 736.34,A -85,B 0,C 180,E1 -11985.375,E2 -11985.375} C_VEL
LIN {X 0,Y 385.303,Z 725.568,A -85,B 0,C 180,E1 -11986.83,E2 -11986.83} C_VEL
LIN {X 0,Y 386.57,Z 713.674,A -85,B 0,C 180,E1 -11988.138,E2 -11988.138} C_VEL
LIN {X 0,Y 387.676,Z 700.748,A -85,B 0,C 180,E1 -11989.291,E2 -11989.291} C_VEL
LIN {X 0,Y 388.78,Z 687.334,A -85,B 0,C 180,E1 -11990.224,E2 -11990.224} C_VEL
LIN {X 0,Y 389.7,Z 673.055,A -85,B 0,C 180,E1 -11990.968,E2 -11990.968} C_VEL
LIN {X 0,Y 390.499,Z 658.964,A -85,B 0,C 180,E1 -11991.476,E2 -11991.476} C_VEL
LIN {X 0,Y 390.99,Z 638.331,A -85,B 0,C 180,E1 -11991.932,E2 -11991.932} C_VEL
LIN {X 0,Y 392.682,Z 550.443,A -85,B 0,C 180,E1 -11993.655,E2 -11993.655} C_VEL
LIN {X 0,Y 388.562,Z 522.056,A -85,B 0,C 180,E1 -11994.513,E2 -11994.513} C_VEL
LIN {X 0,Y 390.422,Z 505.448,A -85,B 0,C 180,E1 -11997.322,E2 -11997.322} C_VEL
LIN {X 0,Y 389.986,Z 501.847,A -85,B 0,C 180,E1 -11997.989,E2 -11997.989} C_VEL
LIN {X 0,Y 386.908,Z 488.83,A -85,B 0,C 180,E1 -12000.569,E2 -12000.569} C_VEL
LIN {X 0,Y 383.042,Z 474.387,A -85,B 0,C 180,E1 -12003.628,E2 -12003.628} C_VEL
LIN {X 0,Y 382.993,Z 474.404,A -85,B 0,C 180,E1 -12007.267,E2 -12007.267} C_VEL
LIN {X 0,Y 383.015,Z 474.4,A -85,B 0,C 180,E1 -12009.955,E2 -12009.955} C_VEL
LIN {X 0,Y 383.058,Z 474.397,A -85,B 0,C 180,E1 -12012.787,E2 -12012.787} C_VEL
LIN {X 0,Y 383.064,Z 474.39,A -85,B 0,C 180,E1 -12015.799,E2 -12015.799} C_VEL
LIN {X 0,Y 383.036,Z 474.397,A -85,B 0,C 180,E1 -12018.785,E2 -12018.785} C_VEL
LIN {X 0,Y 382.994,Z 474.398,A -85,B 0,C 180,E1 -12022.094,E2 -12022.094} C_VEL
LIN {X 0,Y 383.009,Z 474.389,A -85,B 0,C 180,E1 -12025.331,E2 -12025.331} C_VEL
LIN {X 0,Y 383.027,Z 474.394,A -85,B 0,C 180,E1 -12027.852,E2 -12027.852} C_VEL
LIN {X 0,Y 383.053,Z 474.39,A -85,B 0,C 180,E1 -12031.72,E2 -12031.72} C_VEL
LIN {X 0,Y 383.041,Z 474.392,A -85,B 0,C 180,E1 -12035.039,E2 -12035.039} C_VEL
LIN {X 0,Y 382.982,Z 474.377,A -85,B 0,C 180,E1 -12038.468,E2 -12038.468} C_VEL
LIN {X 0,Y 383.052,Z 474.393,A -85,B 0,C 180,E1 -12041.826,E2 -12041.826} C_VEL
LIN {X 0,Y 383.101,Z 474.387,A -85,B 0,C 180,E1 -12045.118,E2 -12045.118} C_VEL
LIN {X 0,Y 383.098,Z 474.385,A -85,B 0,C 180,E1 -12048.358,E2 -12048.358} C_VEL
LIN {X 0,Y 383.292,Z 474.364,A -85,B 0,C 180,E1 -12051.933,E2 -12051.933} C_VEL
LIN {X 0,Y 383.191,Z 474.376,A -85,B 0,C 180,E1 -12054.739,E2 -12054.739} C_VEL
LIN {X 0,Y 383.377,Z 474.349,A -85,B 0,C 180,E1 -12057.899,E2 -12057.899} C_VEL
LIN {X 0,Y 383.51,Z 474.334,A -85,B 0,C 180,E1 -12060,E2 -12060} C_VEL
LIN {X 0,Y 383.242,Z 474.361,A -85,B 0,C 180,E1 -12063.154,E2 -12063.154} C_VEL
LIN {X 0,Y 383.258,Z 474.367,A -85,B 0,C 180,E1 -12066.647,E2 -12066.647} C_VEL
LIN {X 0,Y 383.249,Z 474.364,A -85,B 0,C 180,E1 -12068.436,E2 -12068.436} C_VEL
LIN {X 0,Y 383.097,Z 474.387,A -85,B 0,C 180,E1 -12071.642,E2 -12071.642} C_VEL
LIN {X 0,Y 383.104,Z 474.39,A -85,B 0,C 180,E1 -12074.882,E2 -12074.882} C_VEL
LIN {X 0,Y 383.079,Z 474.385,A -85,B 0,C 180,E1 -12078.173,E2 -12078.173} C_VEL
LIN {X 0,Y 382.986,Z 474.398,A -85,B 0,C 180,E1 -12081.532,E2 -12081.532} C_VEL
LIN {X 0,Y 383.043,Z 474.394,A -85,B 0,C 180,E1 -12084.961,E2 -12084.961} C_VEL
LIN {X 0,Y 383.04,Z 474.399,A -85,B 0,C 180,E1 -12088.493,E2 -12088.493} C_VEL
LIN {X 0,Y 383.018,Z 474.402,A -85,B 0,C 180,E1 -12092.433,E2 -12092.433} C_VEL
LIN {X 0,Y 383.026,Z 474.4,A -85,B 0,C 180,E1 -12096.166,E2 -12096.166} C_VEL
LIN {X 0,Y 383.012,Z 474.4,A -85,B 0,C 180,E1 -12099.958,E2 -12099.958} C_VEL
LIN {X 0,Y 383.025,Z 474.397,A -85,B 0,C 180,E1 -12102.784,E2 -12102.784} C_VEL
LIN {X 0,Y 383.034,Z 474.395,A -85,B 0,C 180,E1 -12105.797,E2 -12105.797} C_VEL
LIN {X 0,Y 383.039,Z 474.399,A -85,B 0,C 180,E1 -12108.788,E2 -12108.788} C_VEL
LIN {X 0,Y 382.999,Z 474.398,A -85,B 0,C 180,E1 -12112.097,E2 -12112.097} C_VEL
LIN {X 0,Y 383.014,Z 474.399,A -85,B 0,C 180,E1 -12115.334,E2 -12115.334} C_VEL
LIN {X 0,Y 383.017,Z 474.468,A -85,B 0,C 180,E1 -12118.914,E2 -12118.914} C_VEL
LIN {X 0,Y 386.09,Z 486.906,A -85,B 0,C 180,E1 -12122.05,E2 -12122.05} C_VEL
LIN {X 0,Y 388.257,Z 497.661,A -85,B 0,C 180,E1 -12124.625,E2 -12124.625} C_VEL
LIN {X 0,Y 388.261,Z 501.187,A -85,B 0,C 180,E1 -12125.399,E2 -12125.399} C_VEL
LIN {X 0,Y 386.857,Z 516.468,A -85,B 0,C 180,E1 -12128.563,E2 -12128.563} C_VEL
LIN {X 0,Y 391.981,Z 542.68,A -85,B 0,C 180,E1 -12129.366,E2 -12129.366} C_VEL
LIN {X 0,Y 390.951,Z 630.419,A -85,B 0,C 180,E1 -12130.884,E2 -12130.884} C_VEL
LIN {X 0,Y 390.477,Z 643.896,A -85,B 0,C 180,E1 -12131.337,E2 -12131.337} C_VEL
LIN {X 0,Y 389.772,Z 656.1,A -85,B 0,C 180,E1 -12131.948,E2 -12131.948} C_VEL
LIN {X 0,Y 388.976,Z 668.36,A -85,B 0,C 180,E1 -12132.792,E2 -12132.792} C_VEL
LIN {X 0,Y 388.163,Z 677.521,A -85,B 0,C 180,E1 -12133.591,E2 -12133.591} C_VEL
LIN {X 0,Y 387.125,Z 688.153,A -85,B 0,C 180,E1 -12134.739,E2 -12134.739} C_VEL
LIN {X 0,Y 386.008,Z 697.86,A -85,B 0,C 180,E1 -12136.042,E2 -12136.042} C_VEL
LIN {X 0,Y 384.905,Z 707.271,A -85,B 0,C 180,E1 -12137.613,E2 -12137.613} C_VEL
LIN {X 0,Y 384.04,Z 714.825,A -85,B 0,C 180,E1 -12139.19,E2 -12139.19} C_VEL
LIN {X 0,Y 383.117,Z 721.77,A -85,B 0,C 180,E1 -12141.031,E2 -12141.031} C_VEL
LIN {X 0,Y 382.56,Z 726.831,A -85,B 0,C 180,E1 -12142.765,E2 -12142.765} C_VEL
LIN {X 0,Y 382.095,Z 731.083,A -85,B 0,C 180,E1 -12144.725,E2 -12144.725} C_VEL
LIN {X 0,Y 382.062,Z 732.748,A -85,B 0,C 180,E1 -12145.782,E2 -12145.782} C_VEL
LIN {X 0,Y 382.011,Z 734.023,A -85,B 0,C 180,E1 -12146.838,E2 -12146.838} C_VEL
LIN {X 0,Y 381.749,Z 735.508,A -85,B 0,C 180,E1 -12148.947,E2 -12148.947} C_VEL
LIN {X 0,Y 381.75,Z 735.548,A -85,B 0,C 180,E1 -12151.056,E2 -12151.056} C_VEL
LIN {X 0,Y 382.003,Z 734.116,A -85,B 0,C 180,E1 -12153.165,E2 -12153.165} C_VEL
LIN {X 0,Y 382.084,Z 731.25,A -85,B 0,C 180,E1 -12155.278,E2 -12155.278} C_VEL
LIN {X 0,Y 382.585,Z 727.004,A -85,B 0,C 180,E1 -12157.265,E2 -12157.265} C_VEL
LIN {X 0,Y 383.105,Z 722.082,A -85,B 0,C 180,E1 -12158.972,E2 -12158.972} C_VEL
LIN {X 0,Y 383.922,Z 715.69,A -85,B 0,C 180,E1 -12160.698,E2 -12160.698} C_VEL
LIN {X 0,Y 383.666,Z 712.577,A -85,B 0,C 180,E1 -12161.446,E2 -12161.446} C_VEL
LIN {X 0,Y 381.571,Z 707.207,A -85,B 0,C 180,E1 -12162.652,E2 -12162.652} C_VEL
LIN {X 0,Y 379.493,Z 701.341,A -85,B 0,C 180,E1 -12163.81,E2 -12163.81} C_VEL
LIN {X 0,Y 379.264,Z 697.321,A -85,B 0,C 180,E1 -12164.47,E2 -12164.47} C_VEL
LIN {X 0,Y 380.463,Z 687.244,A -85,B 0,C 180,E1 -12165.812,E2 -12165.812} C_VEL
LIN {X 0,Y 381.533,Z 676.006,A -85,B 0,C 180,E1 -12167.004,E2 -12167.004} C_VEL
LIN {X 0,Y 382.507,Z 664.98,A -85,B 0,C 180,E1 -12167.925,E2 -12167.925} C_VEL
LIN {X 0,Y 383.429,Z 652.701,A -85,B 0,C 180,E1 -12168.71,E2 -12168.71} C_VEL
LIN {X 0,Y 384.053,Z 639.69,A -85,B 0,C 180,E1 -12169.303,E2 -12169.303} C_VEL
LIN {X 0,Y 384.46,Z 627.091,A -85,B 0,C 180,E1 -12169.663,E2 -12169.663} C_VEL
LIN {X 0,Y 385.443,Z 543.295,A -85,B 0,C 180,E1 -12171.121,E2 -12171.121} C_VEL
LIN {X 0,Y 380.108,Z 516.531,A -85,B 0,C 180,E1 -12171.973,E2 -12171.973} C_VEL
LIN {X 0,Y 381.476,Z 501.822,A -85,B 0,C 180,E1 -12175.072,E2 -12175.072} C_VEL
LIN {X 0,Y 381.354,Z 498.921,A -85,B 0,C 180,E1 -12175.731,E2 -12175.731} C_VEL
LIN {X 0,Y 378.976,Z 487.522,A -85,B 0,C 180,E1 -12178.525,E2 -12178.525} C_VEL
LIN {X 0,Y 376.06,Z 475.79,A -85,B 0,C 180,E1 -12181.554,E2 -12181.554} C_VEL
LIN {X 0,Y 375.969,Z 475.285,A -85,B 0,C 180,E1 -12181.719,E2 -12181.719} C_VEL
LIN {X 0,Y 375.964,Z 475.281,A -85,B 0,C 180,E1 -12185.416,E2 -12185.416} C_VEL
LIN {X 0,Y 375.982,Z 475.272,A -85,B 0,C 180,E1 -12188.272,E2 -12188.272} C_VEL
LIN {X 0,Y 375.942,Z 475.278,A -85,B 0,C 180,E1 -12191.602,E2 -12191.602} C_VEL
LIN {X 0,Y 375.934,Z 475.278,A -85,B 0,C 180,E1 -12195.269,E2 -12195.269} C_VEL
LIN {X 0,Y 375.94,Z 475.276,A -85,B 0,C 180,E1 -12198.4,E2 -12198.4} C_VEL
LIN {X 0,Y 375.98,Z 475.267,A -85,B 0,C 180,E1 -12201.73,E2 -12201.73} C_VEL
LIN {X 0,Y 375.986,Z 475.276,A -85,B 0,C 180,E1 -12205.333,E2 -12205.333} C_VEL
LIN {X 0,Y 375.964,Z 475.278,A -85,B 0,C 180,E1 -12208.438,E2 -12208.438} C_VEL
LIN {X 0,Y 376.004,Z 475.3,A -85,B 0,C 180,E1 -12209.846,E2 -12209.846} C_VEL
LIN {X 0,Y 379.676,Z 491.659,A -85,B 0,C 180,E1 -12212.959,E2 -12212.959} C_VEL
LIN {X 0,Y 380.812,Z 497.443,A -85,B 0,C 180,E1 -12214.033,E2 -12214.033} C_VEL
LIN {X 0,Y 380.039,Z 513.915,A -85,B 0,C 180,E1 -12216.86,E2 -12216.86} C_VEL
LIN {X 0,Y 379.208,Z 530.429,A -85,B 0,C 180,E1 -12219.669,E2 -12219.669} C_VEL
LIN {X 0,Y 382.213,Z 552.254,A -85,B 0,C 180,E1 -12220.343,E2 -12220.343} C_VEL
LIN {X 0,Y 380.13,Z 641.448,A -85,B 0,C 180,E1 -12222.481,E2 -12222.481} C_VEL
LIN {X 0,Y 379.738,Z 654.281,A -85,B 0,C 180,E1 -12222.983,E2 -12222.983} C_VEL
LIN {X 0,Y 379.156,Z 667.361,A -85,B 0,C 180,E1 -12223.718,E2 -12223.718} C_VEL
LIN {X 0,Y 378.457,Z 679.917,A -85,B 0,C 180,E1 -12224.655,E2 -12224.655} C_VEL
LIN {X 0,Y 377.781,Z 691.799,A -85,B 0,C 180,E1 -12225.801,E2 -12225.801} C_VEL
LIN {X 0,Y 377.052,Z 702.382,A -85,B 0,C 180,E1 -12227.075,E2 -12227.075} C_VEL
LIN {X 0,Y 376.375,Z 711.459,A -85,B 0,C 180,E1 -12228.42,E2 -12228.42} C_VEL
LIN {X 0,Y 375.79,Z 720.348,A -85,B 0,C 180,E1 -12230.038,E2 -12230.038} C_VEL
LIN {X 0,Y 375.339,Z 727.404,A -85,B 0,C 180,E1 -12231.656,E2 -12231.656} C_VEL
LIN {X 0,Y 374.977,Z 733.884,A -85,B 0,C 180,E1 -12233.543,E2 -12233.543} C_VEL
LIN {X 0,Y 374.809,Z 738.065,A -85,B 0,C 180,E1 -12235.16,E2 -12235.16} C_VEL
LIN {X 0,Y 374.666,Z 741.133,A -85,B 0,C 180,E1 -12236.774,E2 -12236.774} C_VEL
LIN {X 0,Y 374.657,Z 742.585,A -85,B 0,C 180,E1 -12237.85,E2 -12237.85} C_VEL
LIN {X 0,Y 374.633,Z 743.623,A -85,B 0,C 180,E1 -12238.925,E2 -12238.925} C_VEL
LIN {X 0,Y 374.61,Z 744.224,A -85,B 0,C 180,E1 -12240,E2 -12240} C_VEL
LIN {X 0,Y 374.652,Z 744.363,A -85,B 0,C 180,E1 -12241.075,E2 -12241.075} C_VEL
LIN {X 0,Y 374.754,Z 744.09,A -85,B 0,C 180,E1 -12242.149,E2 -12242.149} C_VEL
LIN {X 0,Y 374.907,Z 743.395,A -85,B 0,C 180,E1 -12243.224,E2 -12243.224} C_VEL
LIN {X 0,Y 374.936,Z 742.236,A -85,B 0,C 180,E1 -12244.3,E2 -12244.3} C_VEL
LIN {X 0,Y 375.132,Z 739.685,A -85,B 0,C 180,E1 -12245.914,E2 -12245.914} C_VEL
LIN {X 0,Y 375.548,Z 736.055,A -85,B 0,C 180,E1 -12247.527,E2 -12247.527} C_VEL
LIN {X 0,Y 376.057,Z 731.253,A -85,B 0,C 180,E1 -12249.14,E2 -12249.14} C_VEL
LIN {X 0,Y 376.782,Z 725.168,A -85,B 0,C 180,E1 -12250.75,E2 -12250.75} C_VEL
LIN {X 0,Y 377.421,Z 718.951,A -85,B 0,C 180,E1 -12252.092,E2 -12252.092} C_VEL
LIN {X 0,Y 378.269,Z 711.465,A -85,B 0,C 180,E1 -12253.429,E2 -12253.429} C_VEL
LIN {X 0,Y 379.275,Z 702.331,A -85,B 0,C 180,E1 -12254.761,E2 -12254.761} C_VEL
LIN {X 0,Y 380.406,Z 690.838,A -85,B 0,C 180,E1 -12256.114,E2 -12256.114} C_VEL
LIN {X 0,Y 381.48,Z 678.167,A -85,B 0,C 180,E1 -12257.282,E2 -12257.282} C_VEL
LIN {X 0,Y 382.447,Z 666.169,A -85,B 0,C 180,E1 -12258.134,E2 -12258.134} C_VEL
LIN {X 0,Y 383.192,Z 653.244,A -85,B 0,C 180,E1 -12258.825,E2 -12258.825} C_VEL
LIN {X 0,Y 383.805,Z 639.875,A -85,B 0,C 180,E1 -12259.314,E2 -12259.314} C_VEL
LIN {X 0,Y 386.778,Z 568.508,A -85,B 0,C 180,E1 -12261.248,E2 -12261.248} C_VEL
LIN {X 0,Y 387.455,Z 553.046,A -85,B 0,C 180,E1 -12261.69,E2 -12261.69} C_VEL
LIN {X 0,Y 384.914,Z 539.986,A -85,B 0,C 180,E1 -12262.372,E2 -12262.372} C_VEL
LIN {X 0,Y 383.588,Z 534.266,A -85,B 0,C 180,E1 -12262.722,E2 -12262.722} C_VEL
LIN {X 0,Y 385.597,Z 510.406,A -85,B 0,C 180,E1 -12266.898,E2 -12266.898} C_VEL
LIN {X 0,Y 385.548,Z 506.157,A -85,B 0,C 180,E1 -12267.699,E2 -12267.699} C_VEL
LIN {X 0,Y 384.115,Z 498.787,A -85,B 0,C 180,E1 -12269.303,E2 -12269.303} C_VEL
LIN {X 0,Y 381.684,Z 490.316,A -85,B 0,C 180,E1 -12271.36,E2 -12271.36} C_VEL
LIN {X 0,Y 378.324,Z 481.127,A -85,B 0,C 180,E1 -12273.869,E2 -12273.869} C_VEL
LIN {X 0,Y 375.991,Z 475.275,A -85,B 0,C 180,E1 -12275.659,E2 -12275.659} C_VEL
LIN {X 0,Y 375.969,Z 475.279,A -85,B 0,C 180,E1 -12279.462,E2 -12279.462} C_VEL
LIN {X 0,Y 375.939,Z 475.282,A -85,B 0,C 180,E1 -12283.189,E2 -12283.189} C_VEL
LIN {X 0,Y 375.939,Z 475.281,A -85,B 0,C 180,E1 -12286.81,E2 -12286.81} C_VEL
LIN {X 0,Y 375.965,Z 475.275,A -85,B 0,C 180,E1 -12290.536,E2 -12290.536} C_VEL
LIN {X 0,Y 375.968,Z 475.279,A -85,B 0,C 180,E1 -12293.495,E2 -12293.495} C_VEL
LIN {X 0,Y 376.028,Z 475.47,A -85,B 0,C 180,E1 -12295.894,E2 -12295.894} C_VEL
LIN {X 0,Y 380.044,Z 490.362,A -85,B 0,C 180,E1 -12299.124,E2 -12299.124} C_VEL
LIN {X 0,Y 383.361,Z 504.354,A -85,B 0,C 180,E1 -12301.961,E2 -12301.961} C_VEL
LIN {X 0,Y 383.66,Z 507.163,A -85,B 0,C 180,E1 -12302.49,E2 -12302.49} C_VEL
LIN {X 0,Y 381.849,Z 522.175,A -85,B 0,C 180,E1 -12305.072,E2 -12305.072} C_VEL
LIN {X 0,Y 386.145,Z 551.186,A -85,B 0,C 180,E1 -12305.956,E2 -12305.956} C_VEL
LIN {X 0,Y 383.956,Z 655.922,A -85,B 0,C 180,E1 -12308.066,E2 -12308.066} C_VEL
LIN {X 0,Y 383.238,Z 670.159,A -85,B 0,C 180,E1 -12308.553,E2 -12308.553} C_VEL
LIN {X 0,Y 382.242,Z 684.521,A -85,B 0,C 180,E1 -12309.271,E2 -12309.271} C_VEL
LIN {X 0,Y 381.203,Z 697.213,A -85,B 0,C 180,E1 -12310.118,E2 -12310.118} C_VEL
LIN {X 0,Y 380.192,Z 709.1,A -85,B 0,C 180,E1 -12311.124,E2 -12311.124} C_VEL
LIN {X 0,Y 379.002,Z 720.658,A -85,B 0,C 180,E1 -12312.322,E2 -12312.322} C_VEL
LIN {X 0,Y 377.819,Z 732.25,A -85,B 0,C 180,E1 -12313.797,E2 -12313.797} C_VEL
LIN {X 0,Y 376.783,Z 742.565,A -85,B 0,C 180,E1 -12315.414,E2 -12315.414} C_VEL
LIN {X 0,Y 376.061,Z 751.117,A -85,B 0,C 180,E1 -12317.039,E2 -12317.039} C_VEL
LIN {X 0,Y 375.332,Z 759.271,A -85,B 0,C 180,E1 -12318.933,E2 -12318.933} C_VEL
LIN {X 0,Y 374.877,Z 765.808,A -85,B 0,C 180,E1 -12320.829,E2 -12320.829} C_VEL
LIN {X 0,Y 374.701,Z 770.279,A -85,B 0,C 180,E1 -12322.454,E2 -12322.454} C_VEL
LIN {X 0,Y 374.639,Z 773.374,A -85,B 0,C 180,E1 -12323.851,E2 -12323.851} C_VEL
LIN {X 0,Y 374.595,Z 776.423,A -85,B 0,C 180,E1 -12325.695,E2 -12325.695} C_VEL
LIN {X 0,Y 374.692,Z 778.63,A -85,B 0,C 180,E1 -12327.849,E2 -12327.849} C_VEL
LIN {X 0,Y 374.644,Z 779.365,A -85,B 0,C 180,E1 -12329.999,E2 -12329.999} C_VEL
LIN {X 0,Y 374.692,Z 778.628,A -85,B 0,C 180,E1 -12332.148,E2 -12332.148} C_VEL
LIN {X 0,Y 374.595,Z 776.42,A -85,B 0,C 180,E1 -12334.302,E2 -12334.302} C_VEL
LIN {X 0,Y 374.67,Z 772.715,A -85,B 0,C 180,E1 -12336.461,E2 -12336.461} C_VEL
LIN {X 0,Y 374.807,Z 767.404,A -85,B 0,C 180,E1 -12338.626,E2 -12338.626} C_VEL
LIN {X 0,Y 375.106,Z 762.238,A -85,B 0,C 180,E1 -12340.251,E2 -12340.251} C_VEL
LIN {X 0,Y 375.734,Z 754.814,A -85,B 0,C 180,E1 -12342.146,E2 -12342.146} C_VEL
LIN {X 0,Y 376.344,Z 746.786,A -85,B 0,C 180,E1 -12343.816,E2 -12343.816} C_VEL
LIN {X 0,Y 377.221,Z 737.617,A -85,B 0,C 180,E1 -12345.395,E2 -12345.395} C_VEL
LIN {X 0,Y 378.286,Z 727.234,A -85,B 0,C 180,E1 -12346.874,E2 -12346.874} C_VEL
LIN {X 0,Y 379.513,Z 715.763,A -85,B 0,C 180,E1 -12348.208,E2 -12348.208} C_VEL
LIN {X 0,Y 380.696,Z 703.047,A -85,B 0,C 180,E1 -12349.407,E2 -12349.407} C_VEL
LIN {X 0,Y 381.796,Z 690.36,A -85,B 0,C 180,E1 -12350.355,E2 -12350.355} C_VEL
LIN {X 0,Y 382.782,Z 677.133,A -85,B 0,C 180,E1 -12351.118,E2 -12351.118} C_VEL
LIN {X 0,Y 383.649,Z 663.146,A -85,B 0,C 180,E1 -12351.702,E2 -12351.702} C_VEL
LIN {X 0,Y 384.185,Z 648.537,A -85,B 0,C 180,E1 -12352.094,E2 -12352.094} C_VEL
LIN {X 0,Y 386.129,Z 551.299,A -85,B 0,C 180,E1 -12354.031,E2 -12354.031} C_VEL
LIN {X 0,Y 381.864,Z 522.036,A -85,B 0,C 180,E1 -12354.933,E2 -12354.933} C_VEL
LIN {X 0,Y 383.622,Z 507.091,A -85,B 0,C 180,E1 -12357.508,E2 -12357.508} C_VEL
LIN {X 0,Y 383.066,Z 503.073,A -85,B 0,C 180,E1 -12358.28,E2 -12358.28} C_VEL
LIN {X 0,Y 380.017,Z 490.275,A -85,B 0,C 180,E1 -12360.875,E2 -12360.875} C_VEL
LIN {X 0,Y 375.988,Z 475.257,A -85,B 0,C 180,E1 -12364.141,E2 -12364.141} C_VEL
LIN {X 0,Y 375.949,Z 475.277,A -85,B 0,C 180,E1 -12366.74,E2 -12366.74} C_VEL
LIN {X 0,Y 375.993,Z 475.275,A -85,B 0,C 180,E1 -12369.971,E2 -12369.971} C_VEL
LIN {X 0,Y 375.991,Z 475.273,A -85,B 0,C 180,E1 -12373.755,E2 -12373.755} C_VEL
LIN {X 0,Y 375.991,Z 475.275,A -85,B 0,C 180,E1 -12376.799,E2 -12376.799} C_VEL
LIN {X 0,Y 375.991,Z 475.269,A -85,B 0,C 180,E1 -12380.026,E2 -12380.026} C_VEL
LIN {X 0,Y 375.956,Z 475.26,A -85,B 0,C 180,E1 -12383.494,E2 -12383.494} C_VEL
LIN {X 0,Y 375.951,Z 475.27,A -85,B 0,C 180,E1 -12385.888,E2 -12385.888} C_VEL
LIN {X 0,Y 375.96,Z 475.274,A -85,B 0,C 180,E1 -12389.687,E2 -12389.687} C_VEL
LIN {X 0,Y 375.992,Z 475.27,A -85,B 0,C 180,E1 -12392.141,E2 -12392.141} C_VEL
LIN {X 0,Y 375.996,Z 475.276,A -85,B 0,C 180,E1 -12394.538,E2 -12394.538} C_VEL
LIN {X 0,Y 375.952,Z 475.25,A -85,B 0,C 180,E1 -12398.045,E2 -12398.045} C_VEL
LIN {X 0,Y 375.998,Z 475.272,A -85,B 0,C 180,E1 -12401.473,E2 -12401.473} C_VEL
LIN {X 0,Y 376.049,Z 475.264,A -85,B 0,C 180,E1 -12404.832,E2 -12404.832} C_VEL
LIN {X 0,Y 376.049,Z 475.264,A -85,B 0,C 180,E1 -12408.137,E2 -12408.137} C_VEL
LIN {X 0,Y 376.246,Z 475.241,A -85,B 0,C 180,E1 -12411.877,E2 -12411.877} C_VEL
LIN {X 0,Y 376.163,Z 475.249,A -85,B 0,C 180,E1 -12414.64,E2 -12414.64} C_VEL
LIN {X 0,Y 376.344,Z 475.225,A -85,B 0,C 180,E1 -12417.86,E2 -12417.86} C_VEL
LIN {X 0,Y 376.479,Z 475.21,A -85,B 0,C 180,E1 -12420,E2 -12420} C_VEL
LIN {X 0,Y 376.18,Z 475.24,A -85,B 0,C 180,E1 -12423.213,E2 -12423.213} C_VEL
LIN {X 0,Y 376.222,Z 475.246,A -85,B 0,C 180,E1 -12426.639,E2 -12426.639} C_VEL
LIN {X 0,Y 376.195,Z 475.243,A -85,B 0,C 180,E1 -12428.595,E2 -12428.595} C_VEL
LIN {X 0,Y 376.048,Z 475.266,A -85,B 0,C 180,E1 -12431.864,E2 -12431.864} C_VEL
LIN {X 0,Y 376.052,Z 475.266,A -85,B 0,C 180,E1 -12435.168,E2 -12435.168} C_VEL
LIN {X 0,Y 376.014,Z 475.267,A -85,B 0,C 180,E1 -12438.527,E2 -12438.527} C_VEL
LIN {X 0,Y 375.954,Z 475.275,A -85,B 0,C 180,E1 -12441.955,E2 -12441.955} C_VEL
LIN {X 0,Y 375.996,Z 475.27,A -85,B 0,C 180,E1 -12445.462,E2 -12445.462} C_VEL
LIN {X 0,Y 375.968,Z 475.274,A -85,B 0,C 180,E1 -12449.08,E2 -12449.08} C_VEL
LIN {X 0,Y 375.969,Z 475.275,A -85,B 0,C 180,E1 -12452.827,E2 -12452.827} C_VEL
LIN {X 0,Y 375.95,Z 475.278,A -85,B 0,C 180,E1 -12455.417,E2 -12455.417} C_VEL
LIN {X 0,Y 375.971,Z 475.277,A -85,B 0,C 180,E1 -12458.273,E2 -12458.273} C_VEL
LIN {X 0,Y 375.953,Z 475.28,A -85,B 0,C 180,E1 -12461.607,E2 -12461.607} C_VEL
LIN {X 0,Y 375.974,Z 475.275,A -85,B 0,C 180,E1 -12465.262,E2 -12465.262} C_VEL
LIN {X 0,Y 375.984,Z 475.275,A -85,B 0,C 180,E1 -12468.391,E2 -12468.391} C_VEL
LIN {X 0,Y 375.964,Z 475.277,A -85,B 0,C 180,E1 -12471.914,E2 -12471.914} C_VEL
LIN {X 0,Y 375.976,Z 475.276,A -85,B 0,C 180,E1 -12475.334,E2 -12475.334} C_VEL
LIN {X 0,Y 375.992,Z 475.356,A -85,B 0,C 180,E1 -12478.443,E2 -12478.443} C_VEL
LIN {X 0,Y 378.888,Z 487.067,A -85,B 0,C 180,E1 -12481.471,E2 -12481.471} C_VEL
LIN {X 0,Y 381.03,Z 497.243,A -85,B 0,C 180,E1 -12483.971,E2 -12483.971} C_VEL
LIN {X 0,Y 381.559,Z 501.374,A -85,B 0,C 180,E1 -12484.937,E2 -12484.937} C_VEL
LIN {X 0,Y 380.094,Z 516.643,A -85,B 0,C 180,E1 -12488.138,E2 -12488.138} C_VEL
LIN {X 0,Y 385.423,Z 543.668,A -85,B 0,C 180,E1 -12488.985,E2 -12488.985} C_VEL
LIN {X 0,Y 384.326,Z 630.354,A -85,B 0,C 180,E1 -12490.506,E2 -12490.506} C_VEL
LIN {X 0,Y 383.835,Z 643.946,A -85,B 0,C 180,E1 -12490.967,E2 -12490.967} C_VEL
LIN {X 0,Y 383.074,Z 656.779,A -85,B 0,C 180,E1 -12491.621,E2 -12491.621} C_VEL
LIN {X 0,Y 382.228,Z 668.925,A -85,B 0,C 180,E1 -12492.479,E2 -12492.479} C_VEL
LIN {X 0,Y 381.375,Z 678.309,A -85,B 0,C 180,E1 -12493.316,E2 -12493.316} C_VEL
LIN {X 0,Y 380.316,Z 688.641,A -85,B 0,C 180,E1 -12494.459,E2 -12494.459} C_VEL
LIN {X 0,Y 379.152,Z 698.326,A -85,B 0,C 180,E1 -12495.784,E2 -12495.784} C_VEL
LIN {X 0,Y 377.999,Z 707.721,A -85,B 0,C 180,E1 -12497.383,E2 -12497.383} C_VEL
LIN {X 0,Y 377.092,Z 715.259,A -85,B 0,C 180,E1 -12498.988,E2 -12498.988} C_VEL
LIN {X 0,Y 376.111,Z 722.195,A -85,B 0,C 180,E1 -12500.862,E2 -12500.862} C_VEL
LIN {X 0,Y 375.501,Z 727.518,A -85,B 0,C 180,E1 -12502.735,E2 -12502.735} C_VEL
LIN {X 0,Y 375.045,Z 731.497,A -85,B 0,C 180,E1 -12504.625,E2 -12504.625} C_VEL
LIN {X 0,Y 374.955,Z 734.433,A -85,B 0,C 180,E1 -12506.778,E2 -12506.778} C_VEL
LIN {X 0,Y 374.682,Z 735.916,A -85,B 0,C 180,E1 -12508.927,E2 -12508.927} C_VEL
LIN {X 0,Y 374.682,Z 735.956,A -85,B 0,C 180,E1 -12511.076,E2 -12511.076} C_VEL
LIN {X 0,Y 374.946,Z 734.525,A -85,B 0,C 180,E1 -12513.225,E2 -12513.225} C_VEL
LIN {X 0,Y 375.035,Z 731.661,A -85,B 0,C 180,E1 -12515.378,E2 -12515.378} C_VEL
LIN {X 0,Y 375.525,Z 727.694,A -85,B 0,C 180,E1 -12517.294,E2 -12517.294} C_VEL
LIN {X 0,Y 376.097,Z 722.505,A -85,B 0,C 180,E1 -12519.141,E2 -12519.141} C_VEL
LIN {X 0,Y 377.033,Z 715.643,A -85,B 0,C 180,E1 -12521.016,E2 -12521.016} C_VEL
LIN {X 0,Y 377.96,Z 708.226,A -85,B 0,C 180,E1 -12522.621,E2 -12522.621} C_VEL
LIN {X 0,Y 378.835,Z 700.671,A -85,B 0,C 180,E1 -12523.957,E2 -12523.957} C_VEL
LIN {X 0,Y 379.264,Z 697.321,A -85,B 0,C 180,E1 -12524.47,E2 -12524.47} C_VEL
LIN {X 0,Y 379.055,Z 693.165,A -85,B 0,C 180,E1 -12525.106,E2 -12525.106} C_VEL
LIN {X 0,Y 377.094,Z 686.147,A -85,B 0,C 180,E1 -12526.126,E2 -12526.126} C_VEL
LIN {X 0,Y 375.187,Z 678.72,A -85,B 0,C 180,E1 -12527.076,E2 -12527.076} C_VEL
LIN {X 0,Y 375.031,Z 673.8,A -85,B 0,C 180,E1 -12527.58,E2 -12527.58} C_VEL
LIN {X 0,Y 376.104,Z 661.881,A -85,B 0,C 180,E1 -12528.523,E2 -12528.523} C_VEL
LIN {X 0,Y 376.958,Z 649.56,A -85,B 0,C 180,E1 -12529.256,E2 -12529.256} C_VEL
LIN {X 0,Y 377.57,Z 636.831,A -85,B 0,C 180,E1 -12529.789,E2 -12529.789} C_VEL
LIN {X 0,Y 377.941,Z 623.496,A -85,B 0,C 180,E1 -12530.123,E2 -12530.123} C_VEL
LIN {X 0,Y 378.828,Z 543.939,A -85,B 0,C 180,E1 -12531.528,E2 -12531.528} C_VEL
LIN {X 0,Y 373.336,Z 516.622,A -85,B 0,C 180,E1 -12532.417,E2 -12532.417} C_VEL
LIN {X 0,Y 374.672,Z 503.338,A -85,B 0,C 180,E1 -12535.262,E2 -12535.262} C_VEL
LIN {X 0,Y 374.29,Z 499.405,A -85,B 0,C 180,E1 -12536.185,E2 -12536.185} C_VEL
LIN {X 0,Y 372.054,Z 488.997,A -85,B 0,C 180,E1 -12538.797,E2 -12538.797} C_VEL
LIN {X 0,Y 369.447,Z 478.319,A -85,B 0,C 180,E1 -12541.6,E2 -12541.6} C_VEL
LIN {X 0,Y 368.927,Z 476.159,A -85,B 0,C 180,E1 -12542.236,E2 -12542.236} C_VEL
LIN {X 0,Y 368.935,Z 476.154,A -85,B 0,C 180,E1 -12545.002,E2 -12545.002} C_VEL
LIN {X 0,Y 368.916,Z 476.152,A -85,B 0,C 180,E1 -12548.641,E2 -12548.641} C_VEL
LIN {X 0,Y 368.889,Z 476.16,A -85,B 0,C 180,E1 -12552.01,E2 -12552.01} C_VEL
LIN {X 0,Y 368.887,Z 476.156,A -85,B 0,C 180,E1 -12555.177,E2 -12555.177} C_VEL
LIN {X 0,Y 368.888,Z 476.153,A -85,B 0,C 180,E1 -12558.178,E2 -12558.178} C_VEL
LIN {X 0,Y 368.914,Z 476.15,A -85,B 0,C 180,E1 -12561.36,E2 -12561.36} C_VEL
LIN {X 0,Y 368.943,Z 476.152,A -85,B 0,C 180,E1 -12565.147,E2 -12565.147} C_VEL
LIN {X 0,Y 368.936,Z 476.155,A -85,B 0,C 180,E1 -12569.047,E2 -12569.047} C_VEL
LIN {X 0,Y 368.964,Z 476.229,A -85,B 0,C 180,E1 -12569.565,E2 -12569.565} C_VEL
LIN {X 0,Y 372.672,Z 492.572,A -85,B 0,C 180,E1 -12572.712,E2 -12572.712} C_VEL
LIN {X 0,Y 373.959,Z 499.967,A -85,B 0,C 180,E1 -12574.09,E2 -12574.09} C_VEL
LIN {X 0,Y 372.844,Z 520.342,A -85,B 0,C 180,E1 -12577.62,E2 -12577.62} C_VEL
LIN {X 0,Y 372.313,Z 530.621,A -85,B 0,C 180,E1 -12579.383,E2 -12579.383} C_VEL
LIN {X 0,Y 375.348,Z 552.063,A -85,B 0,C 180,E1 -12580.068,E2 -12580.068} C_VEL
LIN {X 0,Y 373.17,Z 642.024,A -85,B 0,C 180,E1 -12582.285,E2 -12582.285} C_VEL
LIN {X 0,Y 372.751,Z 654.722,A -85,B 0,C 180,E1 -12582.796,E2 -12582.796} C_VEL
LIN {X 0,Y 372.117,Z 668.8,A -85,B 0,C 180,E1 -12583.613,E2 -12583.613} C_VEL
LIN {X 0,Y 371.449,Z 680.293,A -85,B 0,C 180,E1 -12584.499,E2 -12584.499} C_VEL
LIN {X 0,Y 370.725,Z 692.783,A -85,B 0,C 180,E1 -12585.732,E2 -12585.732} C_VEL
LIN {X 0,Y 370.093,Z 701.761,A -85,B 0,C 180,E1 -12586.828,E2 -12586.828} C_VEL
LIN {X 0,Y 369.38,Z 711.018,A -85,B 0,C 180,E1 -12588.198,E2 -12588.198} C_VEL
LIN {X 0,Y 368.77,Z 720.051,A -85,B 0,C 180,E1 -12589.846,E2 -12589.846} C_VEL
LIN {X 0,Y 368.276,Z 727.259,A -85,B 0,C 180,E1 -12591.495,E2 -12591.495} C_VEL
LIN {X 0,Y 367.926,Z 733.837,A -85,B 0,C 180,E1 -12593.419,E2 -12593.419} C_VEL
LIN {X 0,Y 367.748,Z 738.13,A -85,B 0,C 180,E1 -12595.066,E2 -12595.066} C_VEL
LIN {X 0,Y 367.574,Z 741.292,A -85,B 0,C 180,E1 -12596.712,E2 -12596.712} C_VEL
LIN {X 0,Y 367.561,Z 742.798,A -85,B 0,C 180,E1 -12597.808,E2 -12597.808} C_VEL
LIN {X 0,Y 367.55,Z 743.877,A -85,B 0,C 180,E1 -12598.904,E2 -12598.904} C_VEL
LIN {X 0,Y 367.543,Z 744.548,A -85,B 0,C 180,E1 -12600,E2 -12600} C_VEL
LIN {X 0,Y 367.588,Z 744.74,A -85,B 0,C 180,E1 -12601.095,E2 -12601.095} C_VEL
LIN {X 0,Y 367.696,Z 744.506,A -85,B 0,C 180,E1 -12602.191,E2 -12602.191} C_VEL
LIN {X 0,Y 367.854,Z 743.86,A -85,B 0,C 180,E1 -12603.286,E2 -12603.286} C_VEL
LIN {X 0,Y 367.864,Z 742.758,A -85,B 0,C 180,E1 -12604.383,E2 -12604.383} C_VEL
LIN {X 0,Y 367.932,Z 741.21,A -85,B 0,C 180,E1 -12605.48,E2 -12605.48} C_VEL
LIN {X 0,Y 368.478,Z 737.548,A -85,B 0,C 180,E1 -12607.336,E2 -12607.336} C_VEL
LIN {X 0,Y 368.873,Z 733.743,A -85,B 0,C 180,E1 -12608.767,E2 -12608.767} C_VEL
LIN {X 0,Y 369.603,Z 728.211,A -85,B 0,C 180,E1 -12610.407,E2 -12610.407} C_VEL
LIN {X 0,Y 370.444,Z 721.222,A -85,B 0,C 180,E1 -12612.045,E2 -12612.045} C_VEL
LIN {X 0,Y 371.455,Z 712.502,A -85,B 0,C 180,E1 -12613.68,E2 -12613.68} C_VEL
LIN {X 0,Y 372.513,Z 703.592,A -85,B 0,C 180,E1 -12615.035,E2 -12615.035} C_VEL
LIN {X 0,Y 373.738,Z 692.573,A -85,B 0,C 180,E1 -12616.384,E2 -12616.384} C_VEL
LIN {X 0,Y 374.754,Z 681.663,A -85,B 0,C 180,E1 -12617.461,E2 -12617.461} C_VEL
LIN {X 0,Y 375.722,Z 669.496,A -85,B 0,C 180,E1 -12618.4,E2 -12618.4} C_VEL
LIN {X 0,Y 376.675,Z 656.302,A -85,B 0,C 180,E1 -12619.163,E2 -12619.163} C_VEL
LIN {X 0,Y 377.409,Z 642.416,A -85,B 0,C 180,E1 -12619.726,E2 -12619.726} C_VEL
LIN {X 0,Y 381.388,Z 557.049,A -85,B 0,C 180,E1 -12622.142,E2 -12622.142} C_VEL
LIN {X 0,Y 381.349,Z 553.722,A -85,B 0,C 180,E1 -12622.262,E2 -12622.262} C_VEL
LIN {X 0,Y 379.008,Z 541.461,A -85,B 0,C 180,E1 -12622.942,E2 -12622.942} C_VEL
LIN {X 0,Y 377.39,Z 534.773,A -85,B 0,C 180,E1 -12623.373,E2 -12623.373} C_VEL
LIN {X 0,Y 379.412,Z 513.07,A -85,B 0,C 180,E1 -12627.235,E2 -12627.235} C_VEL
LIN {X 0,Y 379.496,Z 509.799,A -85,B 0,C 180,E1 -12627.866,E2 -12627.866} C_VEL
LIN {X 0,Y 378.225,Z 502.537,A -85,B 0,C 180,E1 -12629.498,E2 -12629.498} C_VEL
LIN {X 0,Y 375.935,Z 494.234,A -85,B 0,C 180,E1 -12631.564,E2 -12631.564} C_VEL
LIN {X 0,Y 372.885,Z 485.641,A -85,B 0,C 180,E1 -12633.972,E2 -12633.972} C_VEL
LIN {X 0,Y 370.202,Z 479.361,A -85,B 0,C 180,E1 -12636.051,E2 -12636.051} C_VEL
LIN {X 0,Y 368.915,Z 476.156,A -85,B 0,C 180,E1 -12637.212,E2 -12637.212} C_VEL
LIN {X 0,Y 368.916,Z 476.155,A -85,B 0,C 180,E1 -12640.369,E2 -12640.369} C_VEL
LIN {X 0,Y 368.887,Z 476.158,A -85,B 0,C 180,E1 -12643.615,E2 -12643.615} C_VEL
LIN {X 0,Y 368.89,Z 476.159,A -85,B 0,C 180,E1 -12646.695,E2 -12646.695} C_VEL
LIN {X 0,Y 368.916,Z 476.156,A -85,B 0,C 180,E1 -12649.642,E2 -12649.642} C_VEL
LIN {X 0,Y 368.905,Z 476.158,A -85,B 0,C 180,E1 -12653.143,E2 -12653.143} C_VEL
LIN {X 0,Y 368.973,Z 476.325,A -85,B 0,C 180,E1 -12655.357,E2 -12655.357} C_VEL
LIN {X 0,Y 372.336,Z 488.766,A -85,B 0,C 180,E1 -12658.146,E2 -12658.146} C_VEL
LIN {X 0,Y 375.599,Z 501.751,A -85,B 0,C 180,E1 -12660.888,E2 -12660.888} C_VEL
LIN {X 0,Y 376.882,Z 508.342,A -85,B 0,C 180,E1 -12662.211,E2 -12662.211} C_VEL
LIN {X 0,Y 375.578,Z 519.042,A -85,B 0,C 180,E1 -12664.067,E2 -12664.067} C_VEL
LIN {X 0,Y 376.064,Z 526.968,A -85,B 0,C 180,E1 -12664.735,E2 -12664.735} C_VEL
LIN {X 0,Y 376.395,Z 529.98,A -85,B 0,C 180,E1 -12664.886,E2 -12664.886} C_VEL
LIN {X 0,Y 379.604,Z 552.393,A -85,B 0,C 180,E1 -12665.574,E2 -12665.574} C_VEL
LIN {X 0,Y 377.38,Z 654.793,A -85,B 0,C 180,E1 -12667.663,E2 -12667.663} C_VEL
LIN {X 0,Y 376.63,Z 669.372,A -85,B 0,C 180,E1 -12668.157,E2 -12668.157} C_VEL
LIN {X 0,Y 375.585,Z 683.858,A -85,B 0,C 180,E1 -12668.886,E2 -12668.886} C_VEL
LIN {X 0,Y 374.411,Z 697.683,A -85,B 0,C 180,E1 -12669.827,E2 -12669.827} C_VEL
LIN {X 0,Y 373.294,Z 710.004,A -85,B 0,C 180,E1 -12670.905,E2 -12670.905} C_VEL
LIN {X 0,Y 371.946,Z 722.454,A -85,B 0,C 180,E1 -12672.259,E2 -12672.259} C_VEL
LIN {X 0,Y 370.711,Z 733.607,A -85,B 0,C 180,E1 -12673.76,E2 -12673.76} C_VEL
LIN {X 0,Y 369.681,Z 743.639,A -85,B 0,C 180,E1 -12675.409,E2 -12675.409} C_VEL
LIN {X 0,Y 368.943,Z 751.947,A -85,B 0,C 180,E1 -12677.065,E2 -12677.065} C_VEL
LIN {X 0,Y 368.206,Z 759.884,A -85,B 0,C 180,E1 -12678.995,E2 -12678.995} C_VEL
LIN {X 0,Y 367.832,Z 765.384,A -85,B 0,C 180,E1 -12680.652,E2 -12680.652} C_VEL
LIN {X 0,Y 367.585,Z 771.16,A -85,B 0,C 180,E1 -12682.86,E2 -12682.86} C_VEL
LIN {X 0,Y 367.522,Z 774.35,A -85,B 0,C 180,E1 -12684.512,E2 -12684.512} C_VEL
LIN {X 0,Y 367.522,Z 776.011,A -85,B 0,C 180,E1 -12685.612,E2 -12685.612} C_VEL
LIN {X 0,Y 367.592,Z 778.219,A -85,B 0,C 180,E1 -12687.807,E2 -12687.807} C_VEL
LIN {X 0,Y 367.596,Z 778.774,A -85,B 0,C 180,E1 -12688.903,E2 -12688.903} C_VEL
LIN {X 0,Y 367.595,Z 778.772,A -85,B 0,C 180,E1 -12691.094,E2 -12691.094} C_VEL
LIN {X 0,Y 367.591,Z 778.217,A -85,B 0,C 180,E1 -12692.19,E2 -12692.19} C_VEL
LIN {X 0,Y 367.521,Z 776.007,A -85,B 0,C 180,E1 -12694.385,E2 -12694.385} C_VEL
LIN {X 0,Y 367.573,Z 772.296,A -85,B 0,C 180,E1 -12696.586,E2 -12696.586} C_VEL
LIN {X 0,Y 367.745,Z 766.981,A -85,B 0,C 180,E1 -12698.793,E2 -12698.793} C_VEL
LIN {X 0,Y 368.048,Z 761.806,A -85,B 0,C 180,E1 -12700.45,E2 -12700.45} C_VEL
LIN {X 0,Y 368.689,Z 754.371,A -85,B 0,C 180,E1 -12702.382,E2 -12702.382} C_VEL
LIN {X 0,Y 369.329,Z 746.972,A -85,B 0,C 180,E1 -12703.956,E2 -12703.956} C_VEL
LIN {X 0,Y 370.324,Z 737.152,A -85,B 0,C 180,E1 -12705.689,E2 -12705.689} C_VEL
LIN {X 0,Y 371.365,Z 726.74,A -85,B 0,C 180,E1 -12707.198,E2 -12707.198} C_VEL
LIN {X 0,Y 372.729,Z 715.237,A -85,B 0,C 180,E1 -12708.552,E2 -12708.552} C_VEL
LIN {X 0,Y 373.927,Z 702.474,A -85,B 0,C 180,E1 -12709.772,E2 -12709.772} C_VEL
LIN {X 0,Y 375.077,Z 689.935,A -85,B 0,C 180,E1 -12710.721,E2 -12710.721} C_VEL
LIN {X 0,Y 376.137,Z 676.401,A -85,B 0,C 180,E1 -12711.51,E2 -12711.51} C_VEL
LIN {X 0,Y 377.045,Z 662.239,A -85,B 0,C 180,E1 -12712.102,E2 -12712.102} C_VEL
LIN {X 0,Y 377.606,Z 647.07,A -85,B 0,C 180,E1 -12712.5,E2 -12712.5} C_VEL
LIN {X 0,Y 379.526,Z 551.849,A -85,B 0,C 180,E1 -12714.431,E2 -12714.431} C_VEL
LIN {X 0,Y 375.163,Z 522.069,A -85,B 0,C 180,E1 -12715.357,E2 -12715.357} C_VEL
LIN {X 0,Y 376.838,Z 508.252,A -85,B 0,C 180,E1 -12717.789,E2 -12717.789} C_VEL
LIN {X 0,Y 374.597,Z 497.462,A -85,B 0,C 180,E1 -12719.978,E2 -12719.978} C_VEL
LIN {X 0,Y 370.838,Z 483.061,A -85,B 0,C 180,E1 -12723.091,E2 -12723.091} C_VEL
LIN {X 0,Y 368.928,Z 476.131,A -85,B 0,C 180,E1 -12724.686,E2 -12724.686} C_VEL
LIN {X 0,Y 368.916,Z 476.157,A -85,B 0,C 180,E1 -12727.559,E2 -12727.559} C_VEL
LIN {X 0,Y 368.946,Z 476.154,A -85,B 0,C 180,E1 -12730.363,E2 -12730.363} C_VEL
LIN {X 0,Y 368.965,Z 476.148,A -85,B 0,C 180,E1 -12733.629,E2 -12733.629} C_VEL
LIN {X 0,Y 368.945,Z 476.154,A -85,B 0,C 180,E1 -12736.705,E2 -12736.705} C_VEL
LIN {X 0,Y 368.944,Z 476.147,A -85,B 0,C 180,E1 -12739.634,E2 -12739.634} C_VEL
LIN {X 0,Y 368.894,Z 476.141,A -85,B 0,C 180,E1 -12743.143,E2 -12743.143} C_VEL
LIN {X 0,Y 368.89,Z 476.154,A -85,B 0,C 180,E1 -12746.461,E2 -12746.461} C_VEL
LIN {X 0,Y 368.914,Z 476.155,A -85,B 0,C 180,E1 -12750.31,E2 -12750.31} C_VEL
LIN {X 0,Y 368.971,Z 476.147,A -85,B 0,C 180,E1 -12753.534,E2 -12753.534} C_VEL
LIN {X 0,Y 368.955,Z 476.134,A -85,B 0,C 180,E1 -12756.421,E2 -12756.421} C_VEL
LIN {X 0,Y 368.925,Z 476.143,A -85,B 0,C 180,E1 -12759.947,E2 -12759.947} C_VEL
LIN {X 0,Y 368.964,Z 476.144,A -85,B 0,C 180,E1 -12763.398,E2 -12763.398} C_VEL
LIN {X 0,Y 369.049,Z 476.14,A -85,B 0,C 180,E1 -12766.79,E2 -12766.79} C_VEL
LIN {X 0,Y 369.061,Z 476.134,A -85,B 0,C 180,E1 -12770.132,E2 -12770.132} C_VEL
LIN {X 0,Y 369.177,Z 476.122,A -85,B 0,C 180,E1 -12772.342,E2 -12772.342} C_VEL
LIN {X 0,Y 369.136,Z 476.123,A -85,B 0,C 180,E1 -12774.538,E2 -12774.538} C_VEL
LIN {X 0,Y 369.309,Z 476.101,A -85,B 0,C 180,E1 -12777.819,E2 -12777.819} C_VEL
LIN {X 0,Y 369.449,Z 476.085,A -85,B 0,C 180,E1 -12780,E2 -12780} C_VEL
LIN {X 0,Y 369.308,Z 476.107,A -85,B 0,C 180,E1 -12782.181,E2 -12782.181} C_VEL
LIN {X 0,Y 369.192,Z 476.122,A -85,B 0,C 180,E1 -12786.627,E2 -12786.627} C_VEL
LIN {X 0,Y 369.128,Z 476.123,A -85,B 0,C 180,E1 -12788.761,E2 -12788.761} C_VEL
LIN {X 0,Y 369.003,Z 476.145,A -85,B 0,C 180,E1 -12792.094,E2 -12792.094} C_VEL
LIN {X 0,Y 368.991,Z 476.145,A -85,B 0,C 180,E1 -12795.465,E2 -12795.465} C_VEL
LIN {X 0,Y 368.973,Z 476.148,A -85,B 0,C 180,E1 -12798.894,E2 -12798.894} C_VEL
LIN {X 0,Y 368.923,Z 476.15,A -85,B 0,C 180,E1 -12802.396,E2 -12802.396} C_VEL
LIN {X 0,Y 368.99,Z 476.143,A -85,B 0,C 180,E1 -12805.981,E2 -12805.981} C_VEL
LIN {X 0,Y 368.958,Z 476.149,A -85,B 0,C 180,E1 -12808.815,E2 -12808.815} C_VEL
LIN {X 0,Y 368.913,Z 476.157,A -85,B 0,C 180,E1 -12812.237,E2 -12812.237} C_VEL
LIN {X 0,Y 368.921,Z 476.156,A -85,B 0,C 180,E1 -12815.003,E2 -12815.003} C_VEL
LIN {X 0,Y 368.907,Z 476.161,A -85,B 0,C 180,E1 -12818.643,E2 -12818.643} C_VEL
LIN {X 0,Y 368.903,Z 476.159,A -85,B 0,C 180,E1 -12821.82,E2 -12821.82} C_VEL
LIN {X 0,Y 368.949,Z 476.151,A -85,B 0,C 180,E1 -12825.189,E2 -12825.189} C_VEL
LIN {X 0,Y 368.935,Z 476.153,A -85,B 0,C 180,E1 -12828.187,E2 -12828.187} C_VEL
LIN {X 0,Y 368.909,Z 476.157,A -85,B 0,C 180,E1 -12831.36,E2 -12831.36} C_VEL
LIN {X 0,Y 368.933,Z 476.154,A -85,B 0,C 180,E1 -12835.148,E2 -12835.148} C_VEL
LIN {X 0,Y 368.961,Z 476.271,A -85,B 0,C 180,E1 -12837.958,E2 -12837.958} C_VEL
LIN {X 0,Y 372.003,Z 488.538,A -85,B 0,C 180,E1 -12841.202,E2 -12841.202} C_VEL
LIN {X 0,Y 374.205,Z 498.955,A -85,B 0,C 180,E1 -12843.812,E2 -12843.812} C_VEL
LIN {X 0,Y 374.729,Z 502.89,A -85,B 0,C 180,E1 -12844.745,E2 -12844.745} C_VEL
LIN {X 0,Y 373.336,Z 516.599,A -85,B 0,C 180,E1 -12847.68,E2 -12847.68} C_VEL
LIN {X 0,Y 378.827,Z 544.305,A -85,B 0,C 180,E1 -12848.581,E2 -12848.581} C_VEL
LIN {X 0,Y 377.728,Z 630.281,A -85,B 0,C 180,E1 -12850.116,E2 -12850.116} C_VEL
LIN {X 0,Y 377.26,Z 643.214,A -85,B 0,C 180,E1 -12850.551,E2 -12850.551} C_VEL
LIN {X 0,Y 376.487,Z 656.317,A -85,B 0,C 180,E1 -12851.217,E2 -12851.217} C_VEL
LIN {X 0,Y 375.575,Z 667.852,A -85,B 0,C 180,E1 -12852.017,E2 -12852.017} C_VEL
LIN {X 0,Y 374.608,Z 678.658,A -85,B 0,C 180,E1 -12852.986,E2 -12852.986} C_VEL
LIN {X 0,Y 373.514,Z 689.128,A -85,B 0,C 180,E1 -12854.169,E2 -12854.169} C_VEL
LIN {X 0,Y 372.291,Z 698.792,A -85,B 0,C 180,E1 -12855.516,E2 -12855.516} C_VEL
LIN {X 0,Y 371.096,Z 708.17,A -85,B 0,C 180,E1 -12857.144,E2 -12857.144} C_VEL
LIN {X 0,Y 370.15,Z 715.69,A -85,B 0,C 180,E1 -12858.779,E2 -12858.779} C_VEL
LIN {X 0,Y 369.121,Z 722.619,A -85,B 0,C 180,E1 -12860.688,E2 -12860.688} C_VEL
LIN {X 0,Y 368.445,Z 728.194,A -85,B 0,C 180,E1 -12862.699,E2 -12862.699} C_VEL
LIN {X 0,Y 368,Z 731.911,A -85,B 0,C 180,E1 -12864.522,E2 -12864.522} C_VEL
LIN {X 0,Y 367.88,Z 734.843,A -85,B 0,C 180,E1 -12866.716,E2 -12866.716} C_VEL
LIN {X 0,Y 367.616,Z 736.324,A -85,B 0,C 180,E1 -12868.906,E2 -12868.906} C_VEL
LIN {X 0,Y 367.616,Z 736.364,A -85,B 0,C 180,E1 -12871.097,E2 -12871.097} C_VEL
LIN {X 0,Y 367.87,Z 734.935,A -85,B 0,C 180,E1 -12873.287,E2 -12873.287} C_VEL
LIN {X 0,Y 367.991,Z 732.072,A -85,B 0,C 180,E1 -12875.481,E2 -12875.481} C_VEL
LIN {X 0,Y 368.452,Z 728.418,A -85,B 0,C 180,E1 -12877.309,E2 -12877.309} C_VEL
LIN {X 0,Y 369.108,Z 722.926,A -85,B 0,C 180,E1 -12879.315,E2 -12879.315} C_VEL
LIN {X 0,Y 370.084,Z 716.07,A -85,B 0,C 180,E1 -12881.226,E2 -12881.226} C_VEL
LIN {X 0,Y 371.063,Z 708.666,A -85,B 0,C 180,E1 -12882.86,E2 -12882.86} C_VEL
LIN {X 0,Y 371.983,Z 701.124,A -85,B 0,C 180,E1 -12884.219,E2 -12884.219} C_VEL
LIN {X 0,Y 373.291,Z 690.931,A -85,B 0,C 180,E1 -12885.701,E2 -12885.701} C_VEL
LIN {X 0,Y 374.349,Z 680.558,A -85,B 0,C 180,E1 -12886.918,E2 -12886.918} C_VEL
LIN {X 0,Y 375.031,Z 673.8,A -85,B 0,C 180,E1 -12887.58,E2 -12887.58} C_VEL
LIN {X 0,Y 374.854,Z 668.78,A -85,B 0,C 180,E1 -12888.062,E2 -12888.062} C_VEL
LIN {X 0,Y 372.817,Z 660.464,A -85,B 0,C 180,E1 -12888.839,E2 -12888.839} C_VEL
LIN {X 0,Y 370.77,Z 651.803,A -85,B 0,C 180,E1 -12889.508,E2 -12889.508} C_VEL
LIN {X 0,Y 370.557,Z 646.256,A -85,B 0,C 180,E1 -12889.814,E2 -12889.814} C_VEL
LIN {X 0,Y 371.108,Z 633.472,A -85,B 0,C 180,E1 -12890.293,E2 -12890.293} C_VEL
LIN {X 0,Y 371.445,Z 615.354,A -85,B 0,C 180,E1 -12890.672,E2 -12890.672} C_VEL
LIN {X 0,Y 372.369,Z 545.364,A -85,B 0,C 180,E1 -12891.925,E2 -12891.925} C_VEL
LIN {X 0,Y 366.964,Z 518.41,A -85,B 0,C 180,E1 -12892.825,E2 -12892.825} C_VEL
LIN {X 0,Y 366.651,Z 516.466,A -85,B 0,C 180,E1 -12892.93,E2 -12892.93} C_VEL
LIN {X 0,Y 367.855,Z 504.865,A -85,B 0,C 180,E1 -12895.461,E2 -12895.461} C_VEL
LIN {X 0,Y 367.422,Z 500.892,A -85,B 0,C 180,E1 -12896.407,E2 -12896.407} C_VEL
LIN {X 0,Y 365.218,Z 490.676,A -85,B 0,C 180,E1 -12899.022,E2 -12899.022} C_VEL
LIN {X 0,Y 362.318,Z 478.697,A -85,B 0,C 180,E1 -12902.238,E2 -12902.238} C_VEL
LIN {X 0,Y 361.872,Z 477.035,A -85,B 0,C 180,E1 -12902.737,E2 -12902.737} C_VEL
LIN {X 0,Y 361.874,Z 477.034,A -85,B 0,C 180,E1 -12905.637,E2 -12905.637} C_VEL
LIN {X 0,Y 361.877,Z 477.03,A -85,B 0,C 180,E1 -12909.028,E2 -12909.028} C_VEL
LIN {X 0,Y 361.843,Z 477.038,A -85,B 0,C 180,E1 -12912.829,E2 -12912.829} C_VEL
LIN {X 0,Y 361.826,Z 477.041,A -85,B 0,C 180,E1 -12915.947,E2 -12915.947} C_VEL
LIN {X 0,Y 361.841,Z 477.035,A -85,B 0,C 180,E1 -12919.245,E2 -12919.245} C_VEL
LIN {X 0,Y 361.87,Z 477.026,A -85,B 0,C 180,E1 -12922.777,E2 -12922.777} C_VEL
LIN {X 0,Y 361.862,Z 477.037,A -85,B 0,C 180,E1 -12925.72,E2 -12925.72} C_VEL
LIN {X 0,Y 361.932,Z 477.213,A -85,B 0,C 180,E1 -12929.295,E2 -12929.295} C_VEL
LIN {X 0,Y 365.367,Z 492.315,A -85,B 0,C 180,E1 -12932.233,E2 -12932.233} C_VEL
LIN {X 0,Y 367.008,Z 500.905,A -85,B 0,C 180,E1 -12933.868,E2 -12933.868} C_VEL
LIN {X 0,Y 365.979,Z 519.877,A -85,B 0,C 180,E1 -12937.187,E2 -12937.187} C_VEL
LIN {X 0,Y 365.381,Z 530.765,A -85,B 0,C 180,E1 -12939.077,E2 -12939.077} C_VEL
LIN {X 0,Y 368.467,Z 553.098,A -85,B 0,C 180,E1 -12939.815,E2 -12939.815} C_VEL
LIN {X 0,Y 366.214,Z 642.253,A -85,B 0,C 180,E1 -12942.082,E2 -12942.082} C_VEL
LIN {X 0,Y 365.772,Z 654.897,A -85,B 0,C 180,E1 -12942.601,E2 -12942.601} C_VEL
LIN {X 0,Y 365.136,Z 668.957,A -85,B 0,C 180,E1 -12943.435,E2 -12943.435} C_VEL
LIN {X 0,Y 364.449,Z 680.469,A -85,B 0,C 180,E1 -12944.337,E2 -12944.337} C_VEL
LIN {X 0,Y 363.71,Z 692.973,A -85,B 0,C 180,E1 -12945.594,E2 -12945.594} C_VEL
LIN {X 0,Y 362.969,Z 702.974,A -85,B 0,C 180,E1 -12946.849,E2 -12946.849} C_VEL
LIN {X 0,Y 362.264,Z 712.077,A -85,B 0,C 180,E1 -12948.246,E2 -12948.246} C_VEL
LIN {X 0,Y 361.657,Z 720.997,A -85,B 0,C 180,E1 -12949.927,E2 -12949.927} C_VEL
LIN {X 0,Y 361.178,Z 728.08,A -85,B 0,C 180,E1 -12951.608,E2 -12951.608} C_VEL
LIN {X 0,Y 360.86,Z 733.929,A -85,B 0,C 180,E1 -12953.351,E2 -12953.351} C_VEL
LIN {X 0,Y 360.668,Z 738.147,A -85,B 0,C 180,E1 -12954.969,E2 -12954.969} C_VEL
LIN {X 0,Y 360.487,Z 741.415,A -85,B 0,C 180,E1 -12956.647,E2 -12956.647} C_VEL
LIN {X 0,Y 360.465,Z 743.007,A -85,B 0,C 180,E1 -12957.765,E2 -12957.765} C_VEL
LIN {X 0,Y 360.47,Z 744.133,A -85,B 0,C 180,E1 -12958.883,E2 -12958.883} C_VEL
LIN {X 0,Y 360.461,Z 744.849,A -85,B 0,C 180,E1 -12960,E2 -12960} C_VEL
LIN {X 0,Y 360.526,Z 745.116,A -85,B 0,C 180,E1 -12961.117,E2 -12961.117} C_VEL
LIN {X 0,Y 360.641,Z 744.922,A -85,B 0,C 180,E1 -12962.234,E2 -12962.234} C_VEL
LIN {X 0,Y 360.782,Z 744.321,A -85,B 0,C 180,E1 -12963.35,E2 -12963.35} C_VEL
LIN {X 0,Y 360.795,Z 743.303,A -85,B 0,C 180,E1 -12964.469,E2 -12964.469} C_VEL
LIN {X 0,Y 360.896,Z 741.807,A -85,B 0,C 180,E1 -12965.588,E2 -12965.588} C_VEL
LIN {X 0,Y 361.438,Z 738.418,A -85,B 0,C 180,E1 -12967.393,E2 -12967.393} C_VEL
LIN {X 0,Y 361.906,Z 734.5,A -85,B 0,C 180,E1 -12968.937,E2 -12968.937} C_VEL
LIN {X 0,Y 362.677,Z 729.044,A -85,B 0,C 180,E1 -12970.608,E2 -12970.608} C_VEL
LIN {X 0,Y 363.58,Z 722.221,A -85,B 0,C 180,E1 -12972.276,E2 -12972.276} C_VEL
LIN {X 0,Y 364.662,Z 713.68,A -85,B 0,C 180,E1 -12973.94,E2 -12973.94} C_VEL
LIN {X 0,Y 365.524,Z 706.824,A -85,B 0,C 180,E1 -12975.044,E2 -12975.044} C_VEL
LIN {X 0,Y 366.746,Z 697.068,A -85,B 0,C 180,E1 -12976.348,E2 -12976.348} C_VEL
LIN {X 0,Y 367.841,Z 686.66,A -85,B 0,C 180,E1 -12977.484,E2 -12977.484} C_VEL
LIN {X 0,Y 369.059,Z 673.762,A -85,B 0,C 180,E1 -12978.601,E2 -12978.601} C_VEL
LIN {X 0,Y 370.058,Z 661.415,A -85,B 0,C 180,E1 -12979.412,E2 -12979.412} C_VEL
LIN {X 0,Y 370.958,Z 647.26,A -85,B 0,C 180,E1 -12980.083,E2 -12980.083} C_VEL
LIN {X 0,Y 375.524,Z 555.518,A -85,B 0,C 180,E1 -12982.81,E2 -12982.81} C_VEL
LIN {X 0,Y 372.973,Z 542.12,A -85,B 0,C 180,E1 -12983.599,E2 -12983.599} C_VEL
LIN {X 0,Y 371.326,Z 535.195,A -85,B 0,C 180,E1 -12984.086,E2 -12984.086} C_VEL
LIN {X 0,Y 373.378,Z 514.773,A -85,B 0,C 180,E1 -12987.787,E2 -12987.787} C_VEL
LIN {X 0,Y 373.159,Z 510.726,A -85,B 0,C 180,E1 -12988.647,E2 -12988.647} C_VEL
LIN {X 0,Y 371.658,Z 503.502,A -85,B 0,C 180,E1 -12990.387,E2 -12990.387} C_VEL
LIN {X 0,Y 369.814,Z 496.875,A -85,B 0,C 180,E1 -12992.148,E2 -12992.148} C_VEL
LIN {X 0,Y 367.009,Z 488.763,A -85,B 0,C 180,E1 -12994.569,E2 -12994.569} C_VEL
LIN {X 0,Y 363.912,Z 481.668,A -85,B 0,C 180,E1 -12997.137,E2 -12997.137} C_VEL
LIN {X 0,Y 361.902,Z 477.324,A -85,B 0,C 180,E1 -12999.031,E2 -12999.031} C_VEL
LIN {X 0,Y 361.861,Z 477.035,A -85,B 0,C 180,E1 -12999.163,E2 -12999.163} C_VEL
LIN {X 0,Y 361.841,Z 477.039,A -85,B 0,C 180,E1 -13002.828,E2 -13002.828} C_VEL
LIN {X 0,Y 361.823,Z 477.04,A -85,B 0,C 180,E1 -13005.946,E2 -13005.946} C_VEL
LIN {X 0,Y 361.839,Z 477.035,A -85,B 0,C 180,E1 -13009.244,E2 -13009.244} C_VEL
LIN {X 0,Y 361.867,Z 477.033,A -85,B 0,C 180,E1 -13012.776,E2 -13012.776} C_VEL
LIN {X 0,Y 361.918,Z 477.217,A -85,B 0,C 180,E1 -13014.805,E2 -13014.805} C_VEL
LIN {X 0,Y 365.459,Z 490.199,A -85,B 0,C 180,E1 -13017.795,E2 -13017.795} C_VEL
LIN {X 0,Y 368.629,Z 502.843,A -85,B 0,C 180,E1 -13020.535,E2 -13020.535} C_VEL
LIN {X 0,Y 370.075,Z 509.75,A -85,B 0,C 180,E1 -13021.963,E2 -13021.963} C_VEL
LIN {X 0,Y 369.579,Z 514.468,A -85,B 0,C 180,E1 -13022.768,E2 -13022.768} C_VEL
LIN {X 0,Y 370.546,Z 527.565,A -85,B 0,C 180,E1 -13024.023,E2 -13024.023} C_VEL
LIN {X 0,Y 370.642,Z 535.662,A -85,B 0,C 180,E1 -13024.622,E2 -13024.622} C_VEL
LIN {X 0,Y 373.065,Z 553.543,A -85,B 0,C 180,E1 -13025.175,E2 -13025.175} C_VEL
LIN {X 0,Y 370.757,Z 654.935,A -85,B 0,C 180,E1 -13027.279,E2 -13027.279} C_VEL
LIN {X 0,Y 369.965,Z 669.337,A -85,B 0,C 180,E1 -13027.78,E2 -13027.78} C_VEL
LIN {X 0,Y 368.925,Z 683.197,A -85,B 0,C 180,E1 -13028.486,E2 -13028.486} C_VEL
LIN {X 0,Y 367.777,Z 696.599,A -85,B 0,C 180,E1 -13029.406,E2 -13029.406} C_VEL
LIN {X 0,Y 366.557,Z 709.47,A -85,B 0,C 180,E1 -13030.54,E2 -13030.54} C_VEL
LIN {X 0,Y 365.214,Z 720.842,A -85,B 0,C 180,E1 -13031.776,E2 -13031.776} C_VEL
LIN {X 0,Y 364.04,Z 731.303,A -85,B 0,C 180,E1 -13033.166,E2 -13033.166} C_VEL
LIN {X 0,Y 362.901,Z 741.657,A -85,B 0,C 180,E1 -13034.843,E2 -13034.843} C_VEL
LIN {X 0,Y 362.087,Z 750.234,A -85,B 0,C 180,E1 -13036.53,E2 -13036.53} C_VEL
LIN {X 0,Y 361.322,Z 758.41,A -85,B 0,C 180,E1 -13038.498,E2 -13038.498} C_VEL
LIN {X 0,Y 360.773,Z 764.96,A -85,B 0,C 180,E1 -13040.467,E2 -13040.467} C_VEL
LIN {X 0,Y 360.538,Z 769.44,A -85,B 0,C 180,E1 -13042.156,E2 -13042.156} C_VEL
LIN {X 0,Y 360.457,Z 773.124,A -85,B 0,C 180,E1 -13043.917,E2 -13043.917} C_VEL
LIN {X 0,Y 360.45,Z 775.606,A -85,B 0,C 180,E1 -13045.525,E2 -13045.525} C_VEL
LIN {X 0,Y 360.492,Z 777.81,A -85,B 0,C 180,E1 -13047.764,E2 -13047.764} C_VEL
LIN {X 0,Y 360.531,Z 778.366,A -85,B 0,C 180,E1 -13048.882,E2 -13048.882} C_VEL
LIN {X 0,Y 360.53,Z 778.364,A -85,B 0,C 180,E1 -13051.116,E2 -13051.116} C_VEL
LIN {X 0,Y 360.492,Z 777.806,A -85,B 0,C 180,E1 -13052.233,E2 -13052.233} C_VEL
LIN {X 0,Y 360.45,Z 775.595,A -85,B 0,C 180,E1 -13054.472,E2 -13054.472} C_VEL
LIN {X 0,Y 360.491,Z 771.879,A -85,B 0,C 180,E1 -13056.716,E2 -13056.716} C_VEL
LIN {X 0,Y 360.67,Z 766.557,A -85,B 0,C 180,E1 -13058.967,E2 -13058.967} C_VEL
LIN {X 0,Y 361.01,Z 761.376,A -85,B 0,C 180,E1 -13060.656,E2 -13060.656} C_VEL
LIN {X 0,Y 361.66,Z 753.931,A -85,B 0,C 180,E1 -13062.626,E2 -13062.626} C_VEL
LIN {X 0,Y 362.432,Z 745.982,A -85,B 0,C 180,E1 -13064.338,E2 -13064.338} C_VEL
LIN {X 0,Y 363.421,Z 736.688,A -85,B 0,C 180,E1 -13065.994,E2 -13065.994} C_VEL
LIN {X 0,Y 364.505,Z 726.249,A -85,B 0,C 180,E1 -13067.532,E2 -13067.532} C_VEL
LIN {X 0,Y 365.931,Z 714.71,A -85,B 0,C 180,E1 -13068.909,E2 -13068.909} C_VEL
LIN {X 0,Y 367.205,Z 701.907,A -85,B 0,C 180,E1 -13070.15,E2 -13070.15} C_VEL
LIN {X 0,Y 368.474,Z 688.49,A -85,B 0,C 180,E1 -13071.17,E2 -13071.17} C_VEL
LIN {X 0,Y 369.586,Z 674.367,A -85,B 0,C 180,E1 -13071.984,E2 -13071.984} C_VEL
LIN {X 0,Y 370.53,Z 660.205,A -85,B 0,C 180,E1 -13072.549,E2 -13072.549} C_VEL
LIN {X 0,Y 371.041,Z 643.929,A -85,B 0,C 180,E1 -13072.957,E2 -13072.957} C_VEL
LIN {X 0,Y 372.948,Z 552.41,A -85,B 0,C 180,E1 -13074.844,E2 -13074.844} C_VEL
LIN {X 0,Y 368.5,Z 521.971,A -85,B 0,C 180,E1 -13075.823,E2 -13075.823} C_VEL
LIN {X 0,Y 370.02,Z 509.655,A -85,B 0,C 180,E1 -13078.038,E2 -13078.038} C_VEL
LIN {X 0,Y 367.204,Z 496.804,A -85,B 0,C 180,E1 -13080.728,E2 -13080.728} C_VEL
LIN {X 0,Y 363.175,Z 481.619,A -85,B 0,C 180,E1 -13084.136,E2 -13084.136} C_VEL
LIN {X 0,Y 361.876,Z 477.009,A -85,B 0,C 180,E1 -13085.246,E2 -13085.246} C_VEL
LIN {X 0,Y 361.869,Z 477.03,A -85,B 0,C 180,E1 -13089.026,E2 -13089.026} C_VEL
LIN {X 0,Y 361.879,Z 477.033,A -85,B 0,C 180,E1 -13092.439,E2 -13092.439} C_VEL
LIN {X 0,Y 361.922,Z 477.024,A -85,B 0,C 180,E1 -13095.927,E2 -13095.927} C_VEL
LIN {X 0,Y 361.897,Z 477.026,A -85,B 0,C 180,E1 -13099.231,E2 -13099.231} C_VEL
LIN {X 0,Y 361.864,Z 477.018,A -85,B 0,C 180,E1 -13102.982,E2 -13102.982} C_VEL
LIN {X 0,Y 361.852,Z 477.032,A -85,B 0,C 180,E1 -13106.629,E2 -13106.629} C_VEL
LIN {X 0,Y 361.867,Z 477.03,A -85,B 0,C 180,E1 -13109.671,E2 -13109.671} C_VEL
LIN {X 0,Y 361.944,Z 477.023,A -85,B 0,C 180,E1 -13113.474,E2 -13113.474} C_VEL
LIN {X 0,Y 361.879,Z 477.006,A -85,B 0,C 180,E1 -13117.144,E2 -13117.144} C_VEL
LIN {X 0,Y 361.895,Z 477.026,A -85,B 0,C 180,E1 -13120.723,E2 -13120.723} C_VEL
LIN {X 0,Y 361.921,Z 477.023,A -85,B 0,C 180,E1 -13123.066,E2 -13123.066} C_VEL
LIN {X 0,Y 361.989,Z 477.021,A -85,B 0,C 180,E1 -13126.528,E2 -13126.528} C_VEL
LIN {X 0,Y 362.025,Z 477.009,A -85,B 0,C 180,E1 -13129.938,E2 -13129.938} C_VEL
LIN {X 0,Y 362.14,Z 477,A -85,B 0,C 180,E1 -13132.192,E2 -13132.192} C_VEL
LIN {X 0,Y 362.109,Z 476.996,A -85,B 0,C 180,E1 -13134.431,E2 -13134.431} C_VEL
LIN {X 0,Y 362.273,Z 476.978,A -85,B 0,C 180,E1 -13137.777,E2 -13137.777} C_VEL
LIN {X 0,Y 362.418,Z 476.961,A -85,B 0,C 180,E1 -13140,E2 -13140} C_VEL
LIN {X 0,Y 362.272,Z 476.983,A -85,B 0,C 180,E1 -13142.224,E2 -13142.224} C_VEL
LIN {X 0,Y 362.161,Z 476.997,A -85,B 0,C 180,E1 -13146.687,E2 -13146.687} C_VEL
LIN {X 0,Y 362.064,Z 477.003,A -85,B 0,C 180,E1 -13148.934,E2 -13148.934} C_VEL
LIN {X 0,Y 361.956,Z 477.02,A -85,B 0,C 180,E1 -13152.333,E2 -13152.333} C_VEL
LIN {X 0,Y 361.953,Z 477.021,A -85,B 0,C 180,E1 -13154.621,E2 -13154.621} C_VEL
LIN {X 0,Y 361.949,Z 477.016,A -85,B 0,C 180,E1 -13158.1,E2 -13158.1} C_VEL
LIN {X 0,Y 361.882,Z 477.027,A -85,B 0,C 180,E1 -13161.654,E2 -13161.654} C_VEL
LIN {X 0,Y 361.918,Z 477.024,A -85,B 0,C 180,E1 -13165.291,E2 -13165.291} C_VEL
LIN {X 0,Y 361.913,Z 477.025,A -85,B 0,C 180,E1 -13167.779,E2 -13167.779} C_VEL
LIN {X 0,Y 361.856,Z 477.033,A -85,B 0,C 180,E1 -13171.628,E2 -13171.628} C_VEL
LIN {X 0,Y 361.866,Z 477.033,A -85,B 0,C 180,E1 -13175.346,E2 -13175.346} C_VEL
LIN {X 0,Y 361.868,Z 477.034,A -85,B 0,C 180,E1 -13179.029,E2 -13179.029} C_VEL
LIN {X 0,Y 361.85,Z 477.037,A -85,B 0,C 180,E1 -13182.437,E2 -13182.437} C_VEL
LIN {X 0,Y 361.906,Z 477.027,A -85,B 0,C 180,E1 -13185.933,E2 -13185.933} C_VEL
LIN {X 0,Y 361.9,Z 477.03,A -85,B 0,C 180,E1 -13189.233,E2 -13189.233} C_VEL
LIN {X 0,Y 361.865,Z 477.024,A -85,B 0,C 180,E1 -13192.984,E2 -13192.984} C_VEL
LIN {X 0,Y 361.86,Z 477.029,A -85,B 0,C 180,E1 -13196.631,E2 -13196.631} C_VEL
LIN {X 0,Y 361.88,Z 477.125,A -85,B 0,C 180,E1 -13197.433,E2 -13197.433} C_VEL
LIN {X 0,Y 365.177,Z 490.251,A -85,B 0,C 180,E1 -13200.981,E2 -13200.981} C_VEL
LIN {X 0,Y 367.328,Z 500.449,A -85,B 0,C 180,E1 -13203.589,E2 -13203.589} C_VEL
LIN {X 0,Y 367.914,Z 504.466,A -85,B 0,C 180,E1 -13204.56,E2 -13204.56} C_VEL
LIN {X 0,Y 366.615,Z 516.603,A -85,B 0,C 180,E1 -13207.206,E2 -13207.206} C_VEL
LIN {X 0,Y 372.323,Z 545.328,A -85,B 0,C 180,E1 -13208.175,E2 -13208.175} C_VEL
LIN {X 0,Y 371.15,Z 630.179,A -85,B 0,C 180,E1 -13209.712,E2 -13209.712} C_VEL
LIN {X 0,Y 370.665,Z 643.253,A -85,B 0,C 180,E1 -13210.155,E2 -13210.155} C_VEL
LIN {X 0,Y 369.896,Z 655.855,A -85,B 0,C 180,E1 -13210.797,E2 -13210.797} C_VEL
LIN {X 0,Y 368.865,Z 668.44,A -85,B 0,C 180,E1 -13211.679,E2 -13211.679} C_VEL
LIN {X 0,Y 367.741,Z 680.181,A -85,B 0,C 180,E1 -13212.771,E2 -13212.771} C_VEL
LIN {X 0,Y 366.57,Z 690.662,A -85,B 0,C 180,E1 -13214.004,E2 -13214.004} C_VEL
LIN {X 0,Y 365.427,Z 699.256,A -85,B 0,C 180,E1 -13215.238,E2 -13215.238} C_VEL
LIN {X 0,Y 364.198,Z 708.618,A -85,B 0,C 180,E1 -13216.896,E2 -13216.896} C_VEL
LIN {X 0,Y 363.206,Z 716.121,A -85,B 0,C 180,E1 -13218.562,E2 -13218.562} C_VEL
LIN {X 0,Y 362.145,Z 723.042,A -85,B 0,C 180,E1 -13220.507,E2 -13220.507} C_VEL
LIN {X 0,Y 361.522,Z 727.696,A -85,B 0,C 180,E1 -13222.18,E2 -13222.18} C_VEL
LIN {X 0,Y 361.12,Z 731.309,A -85,B 0,C 180,E1 -13223.857,E2 -13223.857} C_VEL
LIN {X 0,Y 360.823,Z 733.985,A -85,B 0,C 180,E1 -13225.533,E2 -13225.533} C_VEL
LIN {X 0,Y 360.808,Z 735.253,A -85,B 0,C 180,E1 -13226.651,E2 -13226.651} C_VEL
LIN {X 0,Y 360.552,Z 736.732,A -85,B 0,C 180,E1 -13228.885,E2 -13228.885} C_VEL
LIN {X 0,Y 360.552,Z 736.772,A -85,B 0,C 180,E1 -13231.118,E2 -13231.118} C_VEL
LIN {X 0,Y 360.796,Z 735.344,A -85,B 0,C 180,E1 -13233.352,E2 -13233.352} C_VEL
LIN {X 0,Y 360.95,Z 732.482,A -85,B 0,C 180,E1 -13235.588,E2 -13235.588} C_VEL
LIN {X 0,Y 361.406,Z 729.039,A -85,B 0,C 180,E1 -13237.358,E2 -13237.358} C_VEL
LIN {X 0,Y 361.896,Z 725.005,A -85,B 0,C 180,E1 -13238.939,E2 -13238.939} C_VEL
LIN {X 0,Y 362.825,Z 718.652,A -85,B 0,C 180,E1 -13240.888,E2 -13240.888} C_VEL
LIN {X 0,Y 363.749,Z 711.736,A -85,B 0,C 180,E1 -13242.555,E2 -13242.555} C_VEL
LIN {X 0,Y 364.888,Z 703.162,A -85,B 0,C 180,E1 -13244.217,E2 -13244.217} C_VEL
LIN {X 0,Y 366.076,Z 694.391,A -85,B 0,C 180,E1 -13245.593,E2 -13245.593} C_VEL
LIN {X 0,Y 367.351,Z 683.761,A -85,B 0,C 180,E1 -13246.945,E2 -13246.945} C_VEL
LIN {X 0,Y 368.323,Z 674.236,A -85,B 0,C 180,E1 -13247.921,E2 -13247.921} C_VEL
LIN {X 0,Y 369.418,Z 662.493,A -85,B 0,C 180,E1 -13248.871,E2 -13248.871} C_VEL
LIN {X 0,Y 370.308,Z 650.276,A -85,B 0,C 180,E1 -13249.616,E2 -13249.616} C_VEL
LIN {X 0,Y 370.557,Z 646.256,A -85,B 0,C 180,E1 -13249.814,E2 -13249.814} C_VEL
LIN {X 0,Y 370.324,Z 640.62,A -85,B 0,C 180,E1 -13250.085,E2 -13250.085} C_VEL
LIN {X 0,Y 368.049,Z 631.445,A -85,B 0,C 180,E1 -13250.547,E2 -13250.547} C_VEL
LIN {X 0,Y 365.468,Z 622.164,A -85,B 0,C 180,E1 -13250.926,E2 -13250.926} C_VEL
LIN {X 0,Y 364.868,Z 616.357,A -85,B 0,C 180,E1 -13251.073,E2 -13251.073} C_VEL
LIN {X 0,Y 365.892,Z 546.75,A -85,B 0,C 180,E1 -13252.34,E2 -13252.34} C_VEL
LIN {X 0,Y 360.899,Z 521.327,A -85,B 0,C 180,E1 -13253.203,E2 -13253.203} C_VEL
LIN {X 0,Y 359.93,Z 516.586,A -85,B 0,C 180,E1 -13253.404,E2 -13253.404} C_VEL
LIN {X 0,Y 361.06,Z 505.579,A -85,B 0,C 180,E1 -13255.853,E2 -13255.853} C_VEL
LIN {X 0,Y 359.192,Z 495.985,A -85,B 0,C 180,E1 -13258.3,E2 -13258.3} C_VEL
LIN {X 0,Y 356.756,Z 485.615,A -85,B 0,C 180,E1 -13261.089,E2 -13261.089} C_VEL
LIN {X 0,Y 354.841,Z 477.913,A -85,B 0,C 180,E1 -13263.257,E2 -13263.257} C_VEL
LIN {X 0,Y 354.807,Z 477.911,A -85,B 0,C 180,E1 -13266.46,E2 -13266.46} C_VEL
LIN {X 0,Y 354.83,Z 477.911,A -85,B 0,C 180,E1 -13269.424,E2 -13269.424} C_VEL
LIN {X 0,Y 354.795,Z 477.916,A -85,B 0,C 180,E1 -13272.868,E2 -13272.868} C_VEL
LIN {X 0,Y 354.774,Z 477.918,A -85,B 0,C 180,E1 -13276.104,E2 -13276.104} C_VEL
LIN {X 0,Y 354.794,Z 477.912,A -85,B 0,C 180,E1 -13279.179,E2 -13279.179} C_VEL
LIN {X 0,Y 354.814,Z 477.903,A -85,B 0,C 180,E1 -13282.403,E2 -13282.403} C_VEL
LIN {X 0,Y 354.819,Z 477.911,A -85,B 0,C 180,E1 -13284.941,E2 -13284.941} C_VEL
LIN {X 0,Y 354.825,Z 477.912,A -85,B 0,C 180,E1 -13288.785,E2 -13288.785} C_VEL
LIN {X 0,Y 354.901,Z 478.162,A -85,B 0,C 180,E1 -13289.011,E2 -13289.011} C_VEL
LIN {X 0,Y 358.54,Z 494.233,A -85,B 0,C 180,E1 -13292.178,E2 -13292.178} C_VEL
LIN {X 0,Y 360.075,Z 502.088,A -85,B 0,C 180,E1 -13293.682,E2 -13293.682} C_VEL
LIN {X 0,Y 359.278,Z 517.215,A -85,B 0,C 180,E1 -13296.359,E2 -13296.359} C_VEL
LIN {X 0,Y 358.482,Z 531.134,A -85,B 0,C 180,E1 -13298.802,E2 -13298.802} C_VEL
LIN {X 0,Y 361.557,Z 554.258,A -85,B 0,C 180,E1 -13299.569,E2 -13299.569} C_VEL
LIN {X 0,Y 359.227,Z 643.115,A -85,B 0,C 180,E1 -13301.905,E2 -13301.905} C_VEL
LIN {X 0,Y 358.712,Z 656.167,A -85,B 0,C 180,E1 -13302.468,E2 -13302.468} C_VEL
LIN {X 0,Y 358.076,Z 670.003,A -85,B 0,C 180,E1 -13303.319,E2 -13303.319} C_VEL
LIN {X 0,Y 357.313,Z 682.812,A -85,B 0,C 180,E1 -13304.378,E2 -13304.378} C_VEL
LIN {X 0,Y 356.595,Z 694.355,A -85,B 0,C 180,E1 -13305.592,E2 -13305.592} C_VEL
LIN {X 0,Y 355.841,Z 704.148,A -85,B 0,C 180,E1 -13306.872,E2 -13306.872} C_VEL
LIN {X 0,Y 355.138,Z 713.141,A -85,B 0,C 180,E1 -13308.297,E2 -13308.297} C_VEL
LIN {X 0,Y 354.634,Z 720.587,A -85,B 0,C 180,E1 -13309.726,E2 -13309.726} C_VEL
LIN {X 0,Y 354.111,Z 727.858,A -85,B 0,C 180,E1 -13311.439,E2 -13311.439} C_VEL
LIN {X 0,Y 353.782,Z 734.243,A -85,B 0,C 180,E1 -13313.356,E2 -13313.356} C_VEL
LIN {X 0,Y 353.592,Z 738.163,A -85,B 0,C 180,E1 -13314.868,E2 -13314.868} C_VEL
LIN {X 0,Y 353.404,Z 741.531,A -85,B 0,C 180,E1 -13316.58,E2 -13316.58} C_VEL
LIN {X 0,Y 353.369,Z 743.202,A -85,B 0,C 180,E1 -13317.72,E2 -13317.72} C_VEL
LIN {X 0,Y 353.374,Z 744.381,A -85,B 0,C 180,E1 -13318.86,E2 -13318.86} C_VEL
LIN {X 0,Y 353.381,Z 745.141,A -85,B 0,C 180,E1 -13320,E2 -13320} C_VEL
LIN {X 0,Y 353.465,Z 745.487,A -85,B 0,C 180,E1 -13321.139,E2 -13321.139} C_VEL
LIN {X 0,Y 353.587,Z 745.354,A -85,B 0,C 180,E1 -13322.278,E2 -13322.278} C_VEL
LIN {X 0,Y 353.713,Z 744.8,A -85,B 0,C 180,E1 -13323.417,E2 -13323.417} C_VEL
LIN {X 0,Y 353.727,Z 743.845,A -85,B 0,C 180,E1 -13324.558,E2 -13324.558} C_VEL
LIN {X 0,Y 353.862,Z 742.41,A -85,B 0,C 180,E1 -13325.699,E2 -13325.699} C_VEL
LIN {X 0,Y 354.44,Z 739.178,A -85,B 0,C 180,E1 -13327.502,E2 -13327.502} C_VEL
LIN {X 0,Y 354.95,Z 735.287,A -85,B 0,C 180,E1 -13329.114,E2 -13329.114} C_VEL
LIN {X 0,Y 355.939,Z 728.974,A -85,B 0,C 180,E1 -13331.099,E2 -13331.099} C_VEL
LIN {X 0,Y 356.852,Z 722.008,A -85,B 0,C 180,E1 -13332.801,E2 -13332.801} C_VEL
LIN {X 0,Y 358.094,Z 713.308,A -85,B 0,C 180,E1 -13334.491,E2 -13334.491} C_VEL
LIN {X 0,Y 359.291,Z 704.429,A -85,B 0,C 180,E1 -13335.893,E2 -13335.893} C_VEL
LIN {X 0,Y 360.771,Z 693.014,A -85,B 0,C 180,E1 -13337.339,E2 -13337.339} C_VEL
LIN {X 0,Y 361.892,Z 682.68,A -85,B 0,C 180,E1 -13338.396,E2 -13338.396} C_VEL
LIN {X 0,Y 363.019,Z 670.695,A -85,B 0,C 180,E1 -13339.362,E2 -13339.362} C_VEL
LIN {X 0,Y 364.041,Z 658.525,A -85,B 0,C 180,E1 -13340.113,E2 -13340.113} C_VEL
LIN {X 0,Y 364.885,Z 645.639,A -85,B 0,C 180,E1 -13340.69,E2 -13340.69} C_VEL
LIN {X 0,Y 369.767,Z 557.245,A -85,B 0,C 180,E1 -13343.394,E2 -13343.394} C_VEL
LIN {X 0,Y 367.353,Z 544.157,A -85,B 0,C 180,E1 -13344.2,E2 -13344.2} C_VEL
LIN {X 0,Y 365.383,Z 535.725,A -85,B 0,C 180,E1 -13344.829,E2 -13344.829} C_VEL
LIN {X 0,Y 367.43,Z 516.673,A -85,B 0,C 180,E1 -13348.372,E2 -13348.372} C_VEL
LIN {X 0,Y 366.668,Z 510.879,A -85,B 0,C 180,E1 -13349.712,E2 -13349.712} C_VEL
LIN {X 0,Y 364.649,Z 502.291,A -85,B 0,C 180,E1 -13352.001,E2 -13352.001} C_VEL
LIN {X 0,Y 361.731,Z 493.405,A -85,B 0,C 180,E1 -13354.715,E2 -13354.715} C_VEL
LIN {X 0,Y 358.809,Z 486.389,A -85,B 0,C 180,E1 -13357.387,E2 -13357.387} C_VEL
LIN {X 0,Y 357.189,Z 482.829,A -85,B 0,C 180,E1 -13359.022,E2 -13359.022} C_VEL
LIN {X 0,Y 354.86,Z 478.436,A -85,B 0,C 180,E1 -13361.694,E2 -13361.694} C_VEL
LIN {X 0,Y 354.777,Z 477.916,A -85,B 0,C 180,E1 -13362.022,E2 -13362.022} C_VEL
LIN {X 0,Y 354.768,Z 477.917,A -85,B 0,C 180,E1 -13365.493,E2 -13365.493} C_VEL
LIN {X 0,Y 354.792,Z 477.913,A -85,B 0,C 180,E1 -13369.178,E2 -13369.178} C_VEL
LIN {X 0,Y 354.811,Z 477.911,A -85,B 0,C 180,E1 -13372.402,E2 -13372.402} C_VEL
LIN {X 0,Y 354.828,Z 478.008,A -85,B 0,C 180,E1 -13373.189,E2 -13373.189} C_VEL
LIN {X 0,Y 355.879,Z 480.829,A -85,B 0,C 180,E1 -13374.564,E2 -13374.564} C_VEL
LIN {X 0,Y 356.78,Z 484.708,A -85,B 0,C 180,E1 -13375.826,E2 -13375.826} C_VEL
LIN {X 0,Y 360.802,Z 500.256,A -85,B 0,C 180,E1 -13379.366,E2 -13379.366} C_VEL
LIN {X 0,Y 362.116,Z 505.69,A -85,B 0,C 180,E1 -13380.495,E2 -13380.495} C_VEL
LIN {X 0,Y 363.953,Z 512.567,A -85,B 0,C 180,E1 -13381.606,E2 -13381.606} C_VEL
LIN {X 0,Y 364.503,Z 519.969,A -85,B 0,C 180,E1 -13382.434,E2 -13382.434} C_VEL
LIN {X 0,Y 365.067,Z 530.121,A -85,B 0,C 180,E1 -13383.434,E2 -13383.434} C_VEL
LIN {X 0,Y 364.96,Z 542.324,A -85,B 0,C 180,E1 -13384.376,E2 -13384.376} C_VEL
LIN {X 0,Y 366.53,Z 553.823,A -85,B 0,C 180,E1 -13384.742,E2 -13384.742} C_VEL
LIN {X 0,Y 364.159,Z 655.049,A -85,B 0,C 180,E1 -13386.881,E2 -13386.881} C_VEL
LIN {X 0,Y 363.335,Z 669.309,A -85,B 0,C 180,E1 -13387.39,E2 -13387.39} C_VEL
LIN {X 0,Y 362.211,Z 683.668,A -85,B 0,C 180,E1 -13388.141,E2 -13388.141} C_VEL
LIN {X 0,Y 361.007,Z 696.988,A -85,B 0,C 180,E1 -13389.083,E2 -13389.083} C_VEL
LIN {X 0,Y 359.829,Z 708.937,A -85,B 0,C 180,E1 -13390.161,E2 -13390.161} C_VEL
LIN {X 0,Y 358.467,Z 720.346,A -85,B 0,C 180,E1 -13391.421,E2 -13391.421} C_VEL
LIN {X 0,Y 357.205,Z 730.832,A -85,B 0,C 180,E1 -13392.834,E2 -13392.834} C_VEL
LIN {X 0,Y 355.976,Z 741.206,A -85,B 0,C 180,E1 -13394.541,E2 -13394.541} C_VEL
LIN {X 0,Y 355.068,Z 749.792,A -85,B 0,C 180,E1 -13396.258,E2 -13396.258} C_VEL
LIN {X 0,Y 354.311,Z 757.98,A -85,B 0,C 180,E1 -13398.268,E2 -13398.268} C_VEL
LIN {X 0,Y 353.704,Z 764.535,A -85,B 0,C 180,E1 -13400.275,E2 -13400.275} C_VEL
LIN {X 0,Y 353.471,Z 769.027,A -85,B 0,C 180,E1 -13401.998,E2 -13401.998} C_VEL
LIN {X 0,Y 353.342,Z 773.61,A -85,B 0,C 180,E1 -13404.291,E2 -13404.291} C_VEL
LIN {X 0,Y 353.356,Z 775.317,A -85,B 0,C 180,E1 -13405.435,E2 -13405.435} C_VEL
LIN {X 0,Y 353.393,Z 777.407,A -85,B 0,C 180,E1 -13407.719,E2 -13407.719} C_VEL
LIN {X 0,Y 353.466,Z 777.958,A -85,B 0,C 180,E1 -13408.859,E2 -13408.859} C_VEL
LIN {X 0,Y 353.465,Z 777.956,A -85,B 0,C 180,E1 -13411.138,E2 -13411.138} C_VEL
LIN {X 0,Y 353.315,Z 776.469,A -85,B 0,C 180,E1 -13413.42,E2 -13413.42} C_VEL
LIN {X 0,Y 353.357,Z 775.182,A -85,B 0,C 180,E1 -13414.562,E2 -13414.562} C_VEL
LIN {X 0,Y 353.395,Z 771.46,A -85,B 0,C 180,E1 -13416.851,E2 -13416.851} C_VEL
LIN {X 0,Y 353.613,Z 766.134,A -85,B 0,C 180,E1 -13419.147,E2 -13419.147} C_VEL
LIN {X 0,Y 353.99,Z 760.948,A -85,B 0,C 180,E1 -13420.87,E2 -13420.87} C_VEL
LIN {X 0,Y 354.665,Z 753.493,A -85,B 0,C 180,E1 -13422.879,E2 -13422.879} C_VEL
LIN {X 0,Y 355.447,Z 745.881,A -85,B 0,C 180,E1 -13424.553,E2 -13424.553} C_VEL
LIN {X 0,Y 356.539,Z 736.225,A -85,B 0,C 180,E1 -13426.312,E2 -13426.312} C_VEL
LIN {X 0,Y 357.716,Z 725.762,A -85,B 0,C 180,E1 -13427.876,E2 -13427.876} C_VEL
LIN {X 0,Y 359.143,Z 714.186,A -85,B 0,C 180,E1 -13429.281,E2 -13429.281} C_VEL
LIN {X 0,Y 360.52,Z 701.345,A -85,B 0,C 180,E1 -13430.54,E2 -13430.54} C_VEL
LIN {X 0,Y 361.75,Z 688.836,A -85,B 0,C 180,E1 -13431.51,E2 -13431.51} C_VEL
LIN {X 0,Y 362.886,Z 674.948,A -85,B 0,C 180,E1 -13432.337,E2 -13432.337} C_VEL
LIN {X 0,Y 363.868,Z 661.322,A -85,B 0,C 180,E1 -13432.91,E2 -13432.91} C_VEL
LIN {X 0,Y 364.397,Z 645.813,A -85,B 0,C 180,E1 -13433.325,E2 -13433.325} C_VEL
LIN {X 0,Y 366.445,Z 553.356,A -85,B 0,C 180,E1 -13435.261,E2 -13435.261} C_VEL
LIN {X 0,Y 361.845,Z 521.843,A -85,B 0,C 180,E1 -13436.312,E2 -13436.312} C_VEL
LIN {X 0,Y 363.175,Z 512.644,A -85,B 0,C 180,E1 -13437.985,E2 -13437.985} C_VEL
LIN {X 0,Y 362.878,Z 509.405,A -85,B 0,C 180,E1 -13438.641,E2 -13438.641} C_VEL
LIN {X 0,Y 360.108,Z 497.382,A -85,B 0,C 180,E1 -13441.244,E2 -13441.244} C_VEL
LIN {X 0,Y 356.415,Z 483.495,A -85,B 0,C 180,E1 -13444.444,E2 -13444.444} C_VEL
LIN {X 0,Y 354.819,Z 477.892,A -85,B 0,C 180,E1 -13445.814,E2 -13445.814} C_VEL
LIN {X 0,Y 354.817,Z 477.912,A -85,B 0,C 180,E1 -13449.422,E2 -13449.422} C_VEL
LIN {X 0,Y 354.834,Z 477.913,A -85,B 0,C 180,E1 -13452.875,E2 -13452.875} C_VEL
LIN {X 0,Y 354.859,Z 477.904,A -85,B 0,C 180,E1 -13456.118,E2 -13456.118} C_VEL
LIN {X 0,Y 354.848,Z 477.904,A -85,B 0,C 180,E1 -13459.187,E2 -13459.187} C_VEL
LIN {X 0,Y 354.804,Z 477.905,A -85,B 0,C 180,E1 -13462.4,E2 -13462.4} C_VEL
LIN {X 0,Y 354.803,Z 477.894,A -85,B 0,C 180,E1 -13464.94,E2 -13464.94} C_VEL
LIN {X 0,Y 354.805,Z 477.909,A -85,B 0,C 180,E1 -13468.398,E2 -13468.398} C_VEL
LIN {X 0,Y 354.844,Z 477.904,A -85,B 0,C 180,E1 -13471.619,E2 -13471.619} C_VEL
LIN {X 0,Y 354.889,Z 477.903,A -85,B 0,C 180,E1 -13474.172,E2 -13474.172} C_VEL
LIN {X 0,Y 354.819,Z 477.88,A -85,B 0,C 180,E1 -13477.893,E2 -13477.893} C_VEL
LIN {X 0,Y 354.911,Z 477.899,A -85,B 0,C 180,E1 -13481.891,E2 -13481.891} C_VEL
LIN {X 0,Y 354.932,Z 477.896,A -85,B 0,C 180,E1 -13485.98,E2 -13485.98} C_VEL
LIN {X 0,Y 354.972,Z 477.887,A -85,B 0,C 180,E1 -13489.736,E2 -13489.736} C_VEL
LIN {X 0,Y 355.103,Z 477.876,A -85,B 0,C 180,E1 -13492.037,E2 -13492.037} C_VEL
LIN {X 0,Y 355.083,Z 477.87,A -85,B 0,C 180,E1 -13494.321,E2 -13494.321} C_VEL
LIN {X 0,Y 355.236,Z 477.854,A -85,B 0,C 180,E1 -13497.732,E2 -13497.732} C_VEL
LIN {X 0,Y 355.388,Z 477.837,A -85,B 0,C 180,E1 -13500,E2 -13500} C_VEL
LIN {X 0,Y 355.235,Z 477.858,A -85,B 0,C 180,E1 -13502.268,E2 -13502.268} C_VEL
LIN {X 0,Y 355.127,Z 477.871,A -85,B 0,C 180,E1 -13506.82,E2 -13506.82} C_VEL
LIN {X 0,Y 355.006,Z 477.884,A -85,B 0,C 180,E1 -13509.113,E2 -13509.113} C_VEL
LIN {X 0,Y 354.916,Z 477.893,A -85,B 0,C 180,E1 -13512.581,E2 -13512.581} C_VEL
LIN {X 0,Y 354.882,Z 477.905,A -85,B 0,C 180,E1 -13516.097,E2 -13516.097} C_VEL
LIN {X 0,Y 354.896,Z 477.896,A -85,B 0,C 180,E1 -13518.473,E2 -13518.473} C_VEL
LIN {X 0,Y 354.825,Z 477.906,A -85,B 0,C 180,E1 -13522.107,E2 -13522.107} C_VEL
LIN {X 0,Y 354.89,Z 477.9,A -85,B 0,C 180,E1 -13525.828,E2 -13525.828} C_VEL
LIN {X 0,Y 354.845,Z 477.904,A -85,B 0,C 180,E1 -13529.68,E2 -13529.68} C_VEL
LIN {X 0,Y 354.82,Z 477.906,A -85,B 0,C 180,E1 -13533.709,E2 -13533.709} C_VEL
LIN {X 0,Y 354.792,Z 477.914,A -85,B 0,C 180,E1 -13536.461,E2 -13536.461} C_VEL
LIN {X 0,Y 354.816,Z 477.911,A -85,B 0,C 180,E1 -13539.425,E2 -13539.425} C_VEL
LIN {X 0,Y 354.801,Z 477.912,A -85,B 0,C 180,E1 -13542.872,E2 -13542.872} C_VEL
LIN {X 0,Y 354.846,Z 477.907,A -85,B 0,C 180,E1 -13546.119,E2 -13546.119} C_VEL
LIN {X 0,Y 354.851,Z 477.909,A -85,B 0,C 180,E1 -13549.19,E2 -13549.19} C_VEL
LIN {X 0,Y 354.805,Z 477.905,A -85,B 0,C 180,E1 -13552.404,E2 -13552.404} C_VEL
LIN {X 0,Y 354.809,Z 477.915,A -85,B 0,C 180,E1 -13554.943,E2 -13554.943} C_VEL
LIN {X 0,Y 354.837,Z 478.1,A -85,B 0,C 180,E1 -13556.915,E2 -13556.915} C_VEL
LIN {X 0,Y 357.802,Z 489.629,A -85,B 0,C 180,E1 -13560.125,E2 -13560.125} C_VEL
LIN {X 0,Y 360.259,Z 500.646,A -85,B 0,C 180,E1 -13563.029,E2 -13563.029} C_VEL
LIN {X 0,Y 361.093,Z 506.258,A -85,B 0,C 180,E1 -13564.413,E2 -13564.413} C_VEL
LIN {X 0,Y 359.943,Z 516.943,A -85,B 0,C 180,E1 -13566.741,E2 -13566.741} C_VEL
LIN {X 0,Y 365.425,Z 544.181,A -85,B 0,C 180,E1 -13567.682,E2 -13567.682} C_VEL
LIN {X 0,Y 365.902,Z 547.543,A -85,B 0,C 180,E1 -13567.781,E2 -13567.781} C_VEL
LIN {X 0,Y 364.55,Z 631.312,A -85,B 0,C 180,E1 -13569.328,E2 -13569.328} C_VEL
LIN {X 0,Y 364.007,Z 644.84,A -85,B 0,C 180,E1 -13569.813,E2 -13569.813} C_VEL
LIN {X 0,Y 363.148,Z 657.66,A -85,B 0,C 180,E1 -13570.5,E2 -13570.5} C_VEL
LIN {X 0,Y 362.162,Z 669.019,A -85,B 0,C 180,E1 -13571.327,E2 -13571.327} C_VEL
LIN {X 0,Y 360.985,Z 680.695,A -85,B 0,C 180,E1 -13572.438,E2 -13572.438} C_VEL
LIN {X 0,Y 359.768,Z 691.22,A -85,B 0,C 180,E1 -13573.703,E2 -13573.703} C_VEL
LIN {X 0,Y 358.324,Z 701.457,A -85,B 0,C 180,E1 -13575.229,E2 -13575.229} C_VEL
LIN {X 0,Y 357.094,Z 710.405,A -85,B 0,C 180,E1 -13576.92,E2 -13576.92} C_VEL
LIN {X 0,Y 356.087,Z 717.629,A -85,B 0,C 180,E1 -13578.619,E2 -13578.619} C_VEL
LIN {X 0,Y 355.158,Z 723.465,A -85,B 0,C 180,E1 -13580.318,E2 -13580.318} C_VEL
LIN {X 0,Y 354.492,Z 728.114,A -85,B 0,C 180,E1 -13582.024,E2 -13582.024} C_VEL
LIN {X 0,Y 354.094,Z 731.721,A -85,B 0,C 180,E1 -13583.734,E2 -13583.734} C_VEL
LIN {X 0,Y 353.749,Z 734.396,A -85,B 0,C 180,E1 -13585.444,E2 -13585.444} C_VEL
LIN {X 0,Y 353.722,Z 735.664,A -85,B 0,C 180,E1 -13586.584,E2 -13586.584} C_VEL
LIN {X 0,Y 353.49,Z 737.14,A -85,B 0,C 180,E1 -13588.862,E2 -13588.862} C_VEL
LIN {X 0,Y 353.49,Z 737.179,A -85,B 0,C 180,E1 -13591.141,E2 -13591.141} C_VEL
LIN {X 0,Y 353.709,Z 735.754,A -85,B 0,C 180,E1 -13593.419,E2 -13593.419} C_VEL
LIN {X 0,Y 353.914,Z 732.892,A -85,B 0,C 180,E1 -13595.7,E2 -13595.7} C_VEL
LIN {X 0,Y 354.338,Z 729.71,A -85,B 0,C 180,E1 -13597.381,E2 -13597.381} C_VEL
LIN {X 0,Y 354.902,Z 725.422,A -85,B 0,C 180,E1 -13599.117,E2 -13599.117} C_VEL
LIN {X 0,Y 355.861,Z 719.079,A -85,B 0,C 180,E1 -13601.103,E2 -13601.103} C_VEL
LIN {X 0,Y 356.841,Z 712.172,A -85,B 0,C 180,E1 -13602.803,E2 -13602.803} C_VEL
LIN {X 0,Y 358.019,Z 703.611,A -85,B 0,C 180,E1 -13604.496,E2 -13604.496} C_VEL
LIN {X 0,Y 359.271,Z 694.856,A -85,B 0,C 180,E1 -13605.896,E2 -13605.896} C_VEL
LIN {X 0,Y 360.551,Z 684.627,A -85,B 0,C 180,E1 -13607.228,E2 -13607.228} C_VEL
LIN {X 0,Y 361.619,Z 674.76,A -85,B 0,C 180,E1 -13608.265,E2 -13608.265} C_VEL
LIN {X 0,Y 362.748,Z 663.101,A -85,B 0,C 180,E1 -13609.231,E2 -13609.231} C_VEL
LIN {X 0,Y 363.666,Z 650.988,A -85,B 0,C 180,E1 -13609.989,E2 -13609.989} C_VEL
LIN {X 0,Y 364.38,Z 637.699,A -85,B 0,C 180,E1 -13610.574,E2 -13610.574} C_VEL
LIN {X 0,Y 364.806,Z 624.745,A -85,B 0,C 180,E1 -13610.918,E2 -13610.918} C_VEL
LIN {X 0,Y 364.868,Z 616.357,A -85,B 0,C 180,E1 -13611.073,E2 -13611.073} C_VEL
LIN {X 0,Y 364.327,Z 610.548,A -85,B 0,C 180,E1 -13611.22,E2 -13611.22} C_VEL
LIN {X 0,Y 359.394,Z 591.848,A -85,B 0,C 180,E1 -13611.912,E2 -13611.912} C_VEL
LIN {X 0,Y 358.873,Z 586.038,A -85,B 0,C 180,E1 -13612.062,E2 -13612.062} C_VEL
LIN {X 0,Y 359.28,Z 546.909,A -85,B 0,C 180,E1 -13612.805,E2 -13612.805} C_VEL
LIN {X 0,Y 354.369,Z 522.158,A -85,B 0,C 180,E1 -13613.674,E2 -13613.674} C_VEL
LIN {X 0,Y 353.258,Z 516.71,A -85,B 0,C 180,E1 -13613.892,E2 -13613.892} C_VEL
LIN {X 0,Y 354.214,Z 506.856,A -85,B 0,C 180,E1 -13616.136,E2 -13616.136} C_VEL
LIN {X 0,Y 352.02,Z 496.059,A -85,B 0,C 180,E1 -13618.957,E2 -13618.957} C_VEL
LIN {X 0,Y 349.165,Z 484.065,A -85,B 0,C 180,E1 -13622.287,E2 -13622.287} C_VEL
LIN {X 0,Y 347.778,Z 478.79,A -85,B 0,C 180,E1 -13623.831,E2 -13623.831} C_VEL
LIN {X 0,Y 347.772,Z 478.792,A -85,B 0,C 180,E1 -13627.321,E2 -13627.321} C_VEL
LIN {X 0,Y 347.739,Z 478.794,A -85,B 0,C 180,E1 -13630.298,E2 -13630.298} C_VEL
LIN {X 0,Y 347.73,Z 478.794,A -85,B 0,C 180,E1 -13633.409,E2 -13633.409} C_VEL
LIN {X 0,Y 347.732,Z 478.793,A -85,B 0,C 180,E1 -13636.687,E2 -13636.687} C_VEL
LIN {X 0,Y 347.754,Z 478.791,A -85,B 0,C 180,E1 -13640.173,E2 -13640.173} C_VEL
LIN {X 0,Y 347.768,Z 478.782,A -85,B 0,C 180,E1 -13642.68,E2 -13642.68} C_VEL
LIN {X 0,Y 347.755,Z 478.794,A -85,B 0,C 180,E1 -13645.957,E2 -13645.957} C_VEL
LIN {X 0,Y 347.797,Z 478.955,A -85,B 0,C 180,E1 -13648.687,E2 -13648.687} C_VEL
LIN {X 0,Y 351.536,Z 495.131,A -85,B 0,C 180,E1 -13651.913,E2 -13651.913} C_VEL
LIN {X 0,Y 353.182,Z 503.631,A -85,B 0,C 180,E1 -13653.57,E2 -13653.57} C_VEL
LIN {X 0,Y 352.098,Z 522.751,A -85,B 0,C 180,E1 -13656.981,E2 -13656.981} C_VEL
LIN {X 0,Y 351.559,Z 531.384,A -85,B 0,C 180,E1 -13658.507,E2 -13658.507} C_VEL
LIN {X 0,Y 354.676,Z 554.106,A -85,B 0,C 180,E1 -13659.289,E2 -13659.289} C_VEL
LIN {X 0,Y 352.271,Z 642.899,A -85,B 0,C 180,E1 -13661.686,E2 -13661.686} C_VEL
LIN {X 0,Y 351.737,Z 656.121,A -85,B 0,C 180,E1 -13662.259,E2 -13662.259} C_VEL
LIN {X 0,Y 351.096,Z 670.026,A -85,B 0,C 180,E1 -13663.127,E2 -13663.127} C_VEL
LIN {X 0,Y 350.349,Z 681.99,A -85,B 0,C 180,E1 -13664.119,E2 -13664.119} C_VEL
LIN {X 0,Y 349.671,Z 693.265,A -85,B 0,C 180,E1 -13665.3,E2 -13665.3} C_VEL
LIN {X 0,Y 348.9,Z 703.369,A -85,B 0,C 180,E1 -13666.606,E2 -13666.606} C_VEL
LIN {X 0,Y 348.148,Z 712.527,A -85,B 0,C 180,E1 -13668.058,E2 -13668.058} C_VEL
LIN {X 0,Y 347.497,Z 721.507,A -85,B 0,C 180,E1 -13669.807,E2 -13669.807} C_VEL
LIN {X 0,Y 347.016,Z 728.645,A -85,B 0,C 180,E1 -13671.556,E2 -13671.556} C_VEL
LIN {X 0,Y 346.696,Z 734.533,A -85,B 0,C 180,E1 -13673.37,E2 -13673.37} C_VEL
LIN {X 0,Y 346.453,Z 739.432,A -85,B 0,C 180,E1 -13675.346,E2 -13675.346} C_VEL
LIN {X 0,Y 346.325,Z 741.603,A -85,B 0,C 180,E1 -13676.51,E2 -13676.51} C_VEL
LIN {X 0,Y 346.272,Z 743.342,A -85,B 0,C 180,E1 -13677.673,E2 -13677.673} C_VEL
LIN {X 0,Y 346.278,Z 744.617,A -85,B 0,C 180,E1 -13678.837,E2 -13678.837} C_VEL
LIN {X 0,Y 346.287,Z 745.43,A -85,B 0,C 180,E1 -13680,E2 -13680} C_VEL
LIN {X 0,Y 346.388,Z 745.83,A -85,B 0,C 180,E1 -13681.162,E2 -13681.162} C_VEL
LIN {X 0,Y 346.515,Z 745.788,A -85,B 0,C 180,E1 -13682.325,E2 -13682.325} C_VEL
LIN {X 0,Y 346.63,Z 745.28,A -85,B 0,C 180,E1 -13683.487,E2 -13683.487} C_VEL
LIN {X 0,Y 346.66,Z 744.373,A -85,B 0,C 180,E1 -13684.651,E2 -13684.651} C_VEL
LIN {X 0,Y 346.832,Z 743.035,A -85,B 0,C 180,E1 -13685.815,E2 -13685.815} C_VEL
LIN {X 0,Y 347.448,Z 739.988,A -85,B 0,C 180,E1 -13687.623,E2 -13687.623} C_VEL
